C09107=1084.356,267.374,417.952,175.889,23.890,153.904
C09108=1084.350,267.126,417.980,175.886,23.886,153.903
C09109=1084.344,266.878,418.009,175.884,23.883,153.903
C09110=1084.339,266.630,418.037,175.881,23.880,153.903
C09111=1084.333,266.381,418.065,175.878,23.876,153.902
C09112=1084.328,266.133,418.094,175.876,23.873,153.902
C09113=1084.322,265.884,418.122,175.873,23.870,153.902
C09114=1084.317,265.636,418.151,175.870,23.867,153.901
C09115=1084.311,265.388,418.179,175.868,23.863,153.901
C09116=1084.305,265.140,418.207,175.865,23.860,153.901
C09117=1084.299,264.891,418.235,175.862,23.857,153.900
C09118=1084.294,264.643,418.263,175.860,23.854,153.900
C09119=1084.288,264.394,418.291,175.857,23.850,153.900
C09120=1084.283,264.146,418.319,175.854,23.847,153.899
C09121=1084.276,263.898,418.347,175.852,23.844,153.899
C09122=1084.270,263.649,418.376,175.848,23.841,153.899
C09123=1084.261,263.270,418.419,175.844,23.836,153.898
C09124=1084.253,262.891,418.461,175.840,23.831,153.898
C09125=1084.244,262.512,418.504,175.836,23.826,153.897
C09126=1084.234,262.133,418.546,175.831,23.821,153.897
C09127=1084.229,261.884,418.575,175.829,23.818,153.896
C09128=1084.223,261.636,418.603,175.826,23.815,153.896
C09129=1084.217,261.387,418.631,175.823,23.812,153.896
C09130=1084.211,261.140,418.658,175.821,23.809,153.895
C09131=1084.205,260.891,418.687,175.818,23.805,153.895
C09132=1084.200,260.643,418.715,175.816,23.802,153.895
C09133=1084.195,260.394,418.742,175.812,23.799,153.894
C09134=1084.188,260.146,418.770,175.809,23.796,153.894
C09135=1084.183,259.898,418.798,175.807,23.793,153.894
C09136=1084.177,259.649,418.826,175.804,23.790,153.893
C09137=1084.171,259.401,418.853,175.801,23.786,153.893
C09138=1084.165,259.152,418.882,175.799,23.783,153.893
C09139=1084.160,258.904,418.909,175.796,23.780,153.892
C09140=1084.153,258.655,418.937,175.793,23.777,153.892
C09141=1084.148,258.407,418.965,175.791,23.774,153.892
C09142=1084.142,258.159,418.993,175.788,23.770,153.891
C09143=1084.136,257.910,419.020,175.786,23.768,153.891
C09144=1084.131,257.662,419.048,175.782,23.764,153.891
C09145=1084.125,257.413,419.076,175.780,23.761,153.890
C09146=1084.119,257.165,419.102,175.777,23.758,153.890
C09147=1084.114,256.917,419.130,175.774,23.755,153.890
C09148=1084.108,256.668,419.159,175.771,23.751,153.889
C09149=1084.102,256.420,419.185,175.769,23.749,153.889
C09150=1084.097,256.172,419.213,175.766,23.745,153.889
C09151=1084.091,255.923,419.242,175.764,23.742,153.888
C09152=1084.085,255.675,419.268,175.761,23.739,153.888
C09153=1084.080,255.427,419.296,175.758,23.736,153.888
C09154=1084.074,255.177,419.324,175.756,23.732,153.887
C09155=1084.068,254.929,419.351,175.753,23.729,153.887
C09156=1084.063,254.681,419.379,175.750,23.726,153.887
C09157=1084.056,254.432,419.406,175.748,23.723,153.886
C09158=1084.051,254.184,419.434,175.744,23.720,153.886
C09159=1084.046,253.936,419.461,175.742,23.717,153.886
C09160=1084.039,253.687,419.489,175.739,23.713,153.885
C09161=1084.034,253.439,419.516,175.736,23.710,153.885
C09162=1084.028,253.190,419.543,175.734,23.707,153.885
C09163=1084.023,252.942,419.571,175.731,23.703,153.884
C09164=1084.017,252.693,419.598,175.729,23.701,153.884
C09165=1084.011,252.445,419.626,175.726,23.698,153.884
C09166=1084.006,252.196,419.653,175.723,23.694,153.883
C09167=1084.000,251.949,419.681,175.721,23.691,153.883
C09168=1083.994,251.699,419.708,175.718,23.688,153.883
C09169=1083.989,251.451,419.735,175.716,23.685,153.882
C09170=1083.983,251.203,419.763,175.713,23.681,153.882
C09171=1083.978,250.954,419.789,175.710,23.679,153.882
C09172=1083.973,250.706,419.817,175.708,23.675,153.881
C09173=1083.966,250.457,419.844,175.704,23.672,153.881
C09174=1083.961,250.209,419.872,175.702,23.669,153.881
C09175=1083.952,249.827,419.913,175.698,23.664,153.880
C09176=1083.944,249.445,419.955,175.694,23.659,153.880
C09177=1083.935,249.063,419.997,175.690,23.654,153.879
C09178=1083.926,248.682,420.039,175.686,23.649,153.879
C09179=1083.921,248.433,420.066,175.683,23.646,153.878
C09180=1083.915,248.185,420.093,175.681,23.643,153.878
C09181=1083.910,247.936,420.120,175.678,23.640,153.878
C09182=1083.905,247.687,420.147,175.676,23.636,153.877
C09183=1083.899,247.438,420.174,175.673,23.633,153.877
C09184=1083.893,247.190,420.202,175.670,23.630,153.877
C09185=1083.888,246.942,420.229,175.668,23.627,153.876
C09186=1083.882,246.693,420.255,175.665,23.623,153.876
C09187=1083.876,246.445,420.282,175.662,23.621,153.876
C09188=1083.871,246.196,420.309,175.659,23.617,153.875
C09189=1083.865,245.948,420.336,175.657,23.614,153.875
C09190=1083.859,245.699,420.363,175.654,23.611,153.875
C09191=1083.853,245.451,420.390,175.652,23.608,153.874
C09192=1083.848,245.202,420.417,175.649,23.605,153.874
C09193=1083.842,244.953,420.444,175.646,23.602,153.874
C09194=1083.837,244.705,420.470,175.644,23.598,153.873
C09195=1083.831,244.457,420.497,175.641,23.595,153.873
C09196=1083.826,244.208,420.524,175.639,23.592,153.873
C09197=1083.820,243.960,420.551,175.636,23.589,153.872
C09198=1083.814,243.711,420.577,175.634,23.586,153.872
C09199=1083.809,243.463,420.605,175.630,23.583,153.872
C09200=1083.804,243.214,420.631,175.628,23.580,153.871
C09201=1083.797,242.965,420.658,175.625,23.577,153.871
C09202=1083.791,242.717,420.685,175.623,23.573,153.871
C09203=1083.786,242.469,420.712,175.620,23.570,153.870
C09204=1083.780,242.220,420.738,175.618,23.567,153.870
C09205=1083.774,241.971,420.764,175.615,23.564,153.870
C09206=1083.769,241.723,420.791,175.613,23.561,153.869
C09207=1083.764,241.474,420.818,175.610,23.558,153.869
C09208=1083.758,241.226,420.845,175.607,23.555,153.869
C09209=1083.752,240.977,420.871,175.605,23.552,153.869
C09210=1083.746,240.729,420.898,175.602,23.548,153.868
C09211=1083.741,240.480,420.924,175.599,23.546,153.868
C09212=1083.735,240.232,420.951,175.596,23.542,153.868
C09213=1083.729,239.983,420.977,175.594,23.539,153.867
C09214=1083.723,239.735,421.004,175.591,23.536,153.867
C09215=1083.718,239.486,421.030,175.589,23.533,153.867
C09216=1083.712,239.238,421.057,175.586,23.530,153.866
C09217=1083.706,238.989,421.083,175.584,23.527,153.866
C09218=1083.701,238.740,421.109,175.581,23.524,153.866
C09219=1083.695,238.492,421.136,175.579,23.521,153.865
C09220=1083.689,238.244,421.162,175.576,23.517,153.865
C09221=1083.684,237.995,421.188,175.573,23.515,153.865
C09222=1083.678,237.746,421.215,175.571,23.511,153.864
C09223=1083.672,237.498,421.242,175.568,23.508,153.864
C09224=1083.667,237.249,421.268,175.565,23.505,153.864
C09225=1083.661,237.001,421.294,175.563,23.502,153.864
C09226=1083.656,236.752,421.320,175.560,23.499,153.863
C09227=1083.646,236.364,421.361,175.556,23.494,153.863
C09228=1083.638,235.975,421.403,175.552,23.489,153.862
C09229=1083.629,235.586,421.444,175.548,23.485,153.862
C09230=1083.620,235.197,421.484,175.545,23.480,153.861
C09231=1083.614,234.949,421.511,175.542,23.477,153.861
C09232=1083.609,234.700,421.537,175.540,23.474,153.861
C09233=1083.603,234.451,421.563,175.537,23.470,153.860
C09234=1083.597,234.202,421.589,175.534,23.467,153.860
C09235=1083.592,233.953,421.615,175.531,23.464,153.860
C09236=1083.586,233.705,421.642,175.529,23.461,153.859
C09237=1083.580,233.456,421.667,175.526,23.458,153.859
C09238=1083.574,233.208,421.694,175.524,23.455,153.859
C09239=1083.569,232.960,421.720,175.521,23.452,153.858
C09240=1083.564,232.711,421.745,175.519,23.449,153.858
C09241=1083.558,232.462,421.772,175.516,23.446,153.858
C09242=1083.552,232.214,421.797,175.514,23.443,153.858
C09243=1083.546,231.965,421.824,175.511,23.439,153.857
C09244=1083.541,231.716,421.850,175.509,23.436,153.857
C09245=1083.535,231.467,421.876,175.506,23.434,153.857
C09246=1083.530,231.219,421.902,175.504,23.430,153.856
C09247=1083.524,230.971,421.928,175.501,23.427,153.856
C09248=1083.518,230.722,421.954,175.498,23.424,153.856
C09249=1083.513,230.473,421.979,175.496,23.421,153.855
C09250=1083.507,230.225,422.006,175.493,23.418,153.855
C09251=1083.501,229.976,422.031,175.491,23.415,153.855
C09252=1083.496,229.728,422.057,175.488,23.412,153.854
C09253=1083.490,229.479,422.082,175.486,23.409,153.854
C09254=1083.484,229.230,422.108,175.484,23.406,153.854
C09255=1083.479,228.982,422.135,175.481,23.403,153.853
C09256=1083.472,228.733,422.160,175.478,23.400,153.853
C09257=1083.467,228.484,422.186,175.475,23.397,153.853
C09258=1083.461,228.236,422.211,175.473,23.393,153.852
C09259=1083.456,227.987,422.237,175.470,23.390,153.852
C09260=1083.450,227.739,422.262,175.468,23.388,153.852
C09261=1083.444,227.490,422.288,175.465,23.384,153.852
C09262=1083.439,227.241,422.314,175.463,23.381,153.851
C09263=1083.433,226.993,422.340,175.461,23.378,153.851
C09264=1083.427,226.744,422.366,175.458,23.375,153.851
C09265=1083.421,226.496,422.391,175.456,23.372,153.850
C09266=1083.416,226.247,422.417,175.453,23.369,153.850
C09267=1083.410,225.999,422.442,175.450,23.366,153.850
C09268=1083.405,225.750,422.468,175.447,23.363,153.850
C09269=1083.398,225.501,422.493,175.445,23.360,153.849
C09270=1083.393,225.252,422.519,175.443,23.357,153.849
C09271=1083.388,225.004,422.545,175.440,23.354,153.849
C09272=1083.382,224.755,422.570,175.438,23.351,153.848
C09273=1083.376,224.506,422.596,175.435,23.347,153.848
C09274=1083.371,224.258,422.621,175.433,23.345,153.848
C09275=1083.365,224.009,422.647,175.431,23.342,153.847
C09276=1083.359,223.761,422.672,175.428,23.338,153.847
C09277=1083.354,223.512,422.697,175.426,23.335,153.847
C09278=1083.348,223.263,422.723,175.423,23.332,153.846
C09279=1083.339,222.866,422.764,175.419,23.327,153.846
C09280=1083.330,222.468,422.804,175.416,23.323,153.845
C09281=1083.321,222.071,422.845,175.411,23.318,153.845
C09282=1083.313,221.674,422.885,175.407,23.313,153.844
C09283=1083.306,221.425,422.910,175.404,23.309,153.844
C09284=1083.301,221.177,422.935,175.402,23.306,153.844
C09285=1083.295,220.928,422.961,175.399,23.303,153.843
C09286=1083.289,220.679,422.986,175.397,23.301,153.843
C09287=1083.283,220.430,423.011,175.395,23.298,153.843
C09288=1083.278,220.182,423.037,175.392,23.294,153.842
C09289=1083.272,219.933,423.062,175.390,23.291,153.842
C09290=1083.267,219.685,423.086,175.388,23.289,153.842
C09291=1083.261,219.436,423.112,175.385,23.285,153.842
C09292=1083.255,219.187,423.138,175.383,23.282,153.841
C09293=1083.250,218.938,423.162,175.379,23.279,153.841
C09294=1083.244,218.690,423.187,175.377,23.276,153.841
C09295=1083.237,218.441,423.213,175.375,23.273,153.840
C09296=1083.233,218.192,423.237,175.372,23.270,153.840
C09297=1083.227,217.944,423.263,175.370,23.267,153.840
C09298=1083.221,217.696,423.288,175.368,23.264,153.839
C09299=1083.215,217.446,423.312,175.365,23.261,153.839
C09300=1083.210,217.198,423.338,175.363,23.258,153.839
C09301=1083.204,216.949,423.363,175.360,23.255,153.839
C09302=1083.198,216.700,423.388,175.358,23.252,153.838
C09303=1083.193,216.451,423.412,175.355,23.249,153.838
C09304=1083.187,216.203,423.438,175.353,23.245,153.838
C09305=1083.182,215.955,423.463,175.350,23.243,153.837
C09306=1083.176,215.705,423.488,175.348,23.240,153.837
C09307=1083.170,215.457,423.513,175.345,23.237,153.837
C09308=1083.164,215.208,423.537,175.343,23.234,153.836
C09309=1083.159,214.960,423.562,175.341,23.231,153.836
C09310=1083.154,214.710,423.587,175.338,23.228,153.836
C09311=1083.148,214.462,423.612,175.336,23.224,153.835
C09312=1083.142,214.213,423.637,175.334,23.222,153.835
C09313=1083.137,213.965,423.661,175.331,23.218,153.835
C09314=1083.131,213.716,423.687,175.329,23.215,153.834
C09315=1083.126,213.467,423.712,175.327,23.212,153.834
C09316=1083.120,213.218,423.737,175.324,23.209,153.834
C09317=1083.115,212.970,423.761,175.321,23.206,153.834
C09318=1083.109,212.720,423.786,175.318,23.203,153.833
C09319=1083.103,212.473,423.811,175.316,23.200,153.833
C09320=1083.097,212.223,423.835,175.314,23.197,153.833
C09321=1083.092,211.975,423.860,175.311,23.194,153.832
C09322=1083.086,211.726,423.885,175.309,23.191,153.832
C09323=1083.080,211.477,423.909,175.307,23.188,153.832
C09324=1083.075,211.228,423.934,175.304,23.185,153.831
C09325=1083.069,210.980,423.959,175.302,23.181,153.831
C09326=1083.064,210.732,423.983,175.300,23.179,153.831
C09327=1083.058,210.482,424.008,175.297,23.176,153.830
C09328=1083.052,210.234,424.032,175.294,23.173,153.830
C09329=1083.046,209.985,424.057,175.292,23.170,153.830
C09330=1083.041,209.736,424.082,175.290,23.167,153.829
C09331=1083.031,209.343,424.120,175.286,23.162,153.829
C09332=1083.023,208.950,424.159,175.282,23.157,153.829
C09333=1083.014,208.556,424.198,175.279,23.152,153.828
C09334=1083.005,208.163,424.236,175.275,23.148,153.828
C09335=1082.982,207.132,424.336,175.184,23.100,153.830
C09336=1082.976,206.884,424.359,175.181,23.097,153.830
C09337=1082.970,206.635,424.384,175.179,23.095,153.830
C09338=1082.965,206.386,424.408,175.177,23.093,153.830
C09339=1082.959,206.137,424.431,175.174,23.091,153.830
C09340=1082.954,205.889,424.456,175.172,23.089,153.830
C09341=1082.948,205.640,424.480,175.169,23.087,153.830
C09342=1082.943,205.391,424.503,175.167,23.085,153.830
C09343=1082.937,205.142,424.527,175.164,23.083,153.829
C09344=1082.931,204.894,424.551,175.161,23.080,153.829
C09345=1082.926,204.644,424.575,175.159,23.079,153.829
C09346=1082.921,204.396,424.599,175.156,23.076,153.829
C09347=1082.914,204.148,424.623,175.154,23.075,153.829
C09348=1082.909,203.898,424.646,175.152,23.072,153.829
C09349=1082.904,203.649,424.671,175.149,23.070,153.829
C09350=1082.898,203.400,424.694,175.147,23.068,153.829
C09351=1082.893,203.152,424.718,175.144,23.066,153.829
C09352=1082.887,202.903,424.742,175.142,23.064,153.829
C09353=1082.882,202.654,424.765,175.139,23.062,153.829
C09354=1082.875,202.406,424.789,175.136,23.060,153.828
C09355=1082.871,202.157,424.812,175.134,23.058,153.828
C09356=1082.864,201.908,424.836,175.131,23.056,153.828
C09357=1082.859,201.658,424.860,175.129,23.054,153.828
C09358=1082.853,201.410,424.884,175.127,23.052,153.828
C09359=1082.847,201.161,424.906,175.124,23.050,153.828
C09360=1082.842,200.913,424.931,175.122,23.048,153.828
C09361=1082.836,200.664,424.954,175.119,23.046,153.828
C09362=1082.830,200.414,424.978,175.117,23.044,153.828
C09363=1082.824,200.166,425.001,175.115,23.042,153.828
C09364=1082.818,199.917,425.025,175.112,23.040,153.828
C09365=1082.813,199.668,425.048,175.109,23.037,153.828
C09366=1082.808,199.419,425.071,175.106,23.035,153.828
C09367=1082.802,199.171,425.095,175.104,23.033,153.827
C09368=1082.797,198.922,425.119,175.101,23.031,153.827
C09369=1082.791,198.673,425.142,175.099,23.029,153.827
C09370=1082.785,198.425,425.165,175.097,23.027,153.827
C09371=1082.779,198.175,425.189,175.094,23.025,153.827
C09372=1082.773,197.926,425.213,175.092,23.023,153.827
C09373=1082.768,197.677,425.236,175.089,23.021,153.827
C09374=1082.763,197.428,425.259,175.087,23.019,153.827
C09375=1082.756,197.180,425.283,175.085,23.017,153.827
C09376=1082.751,196.931,425.306,175.082,23.015,153.827
C09377=1082.746,196.682,425.329,175.080,23.013,153.827
C09378=1082.740,196.434,425.353,175.077,23.011,153.827
C09379=1082.734,196.185,425.376,175.075,23.009,153.826
C09380=1082.729,195.935,425.400,175.072,23.007,153.826
C09381=1082.723,195.687,425.422,175.070,23.005,153.826
C09382=1082.717,195.438,425.446,175.068,23.003,153.826
C09383=1082.712,195.189,425.469,175.065,23.001,153.826
C09384=1082.707,194.940,425.493,175.063,22.999,153.826
C09385=1082.701,194.691,425.516,175.060,22.997,153.826
C09386=1082.695,194.443,425.539,175.057,22.994,153.826
C09387=1082.690,194.194,425.563,175.055,22.992,153.826
C09388=1082.684,193.945,425.586,175.052,22.990,153.826
C09389=1082.678,193.696,425.609,175.050,22.988,153.826
C09390=1082.673,193.447,425.632,175.048,22.986,153.825
C09391=1082.668,193.198,425.655,175.045,22.984,153.825
C09392=1082.662,192.950,425.679,175.043,22.982,153.825
C09393=1082.656,192.701,425.702,175.040,22.980,153.825
C09394=1082.650,192.452,425.725,175.038,22.978,153.825
C09395=1082.645,192.203,425.748,175.036,22.976,153.825
C09396=1082.638,191.924,425.773,175.033,22.974,153.825
C09397=1082.632,191.645,425.800,175.031,22.972,153.825
C09398=1082.626,191.366,425.825,175.028,22.969,153.825
C09399=1082.620,191.087,425.851,175.025,22.967,153.825
C09400=1082.614,190.838,425.874,175.023,22.965,153.825
C09401=1082.609,190.589,425.898,175.020,22.963,153.824
C09402=1082.604,190.340,425.920,175.018,22.961,153.824
C09403=1082.598,190.091,425.943,175.016,22.959,153.824
C09404=1082.592,189.842,425.966,175.013,22.956,153.824
C09405=1082.587,189.594,425.989,175.011,22.955,153.824
C09406=1082.582,189.344,426.012,175.008,22.952,153.824
C09407=1082.576,189.096,426.035,175.006,22.950,153.824
C09408=1082.571,188.847,426.058,175.004,22.948,153.824
C09409=1082.565,188.598,426.081,175.001,22.946,153.824
C09410=1082.559,188.349,426.104,174.999,22.944,153.823
C09411=1082.554,188.100,426.128,174.996,22.942,153.823
C09412=1082.549,187.851,426.150,174.994,22.940,153.823
C09413=1082.543,187.603,426.173,174.992,22.938,153.823
C09414=1082.537,187.354,426.196,174.989,22.936,153.823
C09415=1082.532,187.105,426.219,174.987,22.934,153.823
C09416=1082.526,186.856,426.242,174.984,22.932,153.823
C09417=1082.521,186.607,426.264,174.982,22.929,153.823
C09418=1082.516,186.358,426.288,174.980,22.927,153.823
C09419=1082.510,186.109,426.311,174.977,22.925,153.823
C09420=1082.505,185.860,426.333,174.975,22.923,153.823
C09421=1082.499,185.611,426.356,174.973,22.921,153.822
C09422=1082.494,185.363,426.379,174.970,22.919,153.822
C09423=1082.488,185.113,426.401,174.968,22.917,153.822
C09424=1082.483,184.865,426.424,174.966,22.915,153.822
C09425=1082.477,184.616,426.447,174.964,22.913,153.822
C09426=1082.471,184.367,426.470,174.962,22.911,153.822
C09427=1082.466,184.117,426.492,174.959,22.909,153.822
C09428=1082.459,183.869,426.515,174.957,22.907,153.822
C09429=1082.454,183.620,426.537,174.954,22.905,153.822
C09430=1082.449,183.372,426.560,174.952,22.903,153.822
C09431=1082.443,183.122,426.582,174.949,22.901,153.822
C09432=1082.437,182.873,426.605,174.947,22.899,153.822
C09433=1082.431,182.625,426.628,174.945,22.897,153.821
C09434=1082.425,182.375,426.650,174.942,22.895,153.821
C09435=1082.420,182.126,426.673,174.940,22.893,153.821
C09436=1082.414,181.878,426.695,174.937,22.891,153.821
C09437=1082.408,181.629,426.717,174.935,22.889,153.821
C09438=1082.403,181.380,426.740,174.933,22.887,153.821
C09439=1082.397,181.131,426.763,174.931,22.885,153.821
C09440=1082.391,180.882,426.785,174.929,22.884,153.821
C09441=1082.385,180.633,426.808,174.926,22.881,153.821
C09442=1082.380,180.384,426.829,174.924,22.880,153.821
C09443=1082.374,180.135,426.852,174.921,22.877,153.821
C09444=1082.368,179.886,426.874,174.919,22.875,153.821
C09445=1082.363,179.637,426.897,174.917,22.873,153.820
C09446=1082.357,179.388,426.920,174.914,22.871,153.820
C09447=1082.351,179.140,426.941,174.912,22.869,153.820
C09448=1082.346,178.891,426.964,174.909,22.867,153.820
C09449=1082.340,178.641,426.986,174.907,22.865,153.820
C09450=1082.334,178.393,427.009,174.905,22.864,153.820
C09451=1082.329,178.144,427.031,174.903,22.861,153.820
C09452=1082.323,177.895,427.054,174.901,22.860,153.820
C09453=1082.317,177.646,427.075,174.898,22.857,153.820
C09454=1082.311,177.397,427.098,174.896,22.856,153.820
C09455=1082.306,177.148,427.120,174.893,22.853,153.820
C09456=1082.300,176.899,427.142,174.891,22.851,153.819
C09457=1082.295,176.650,427.165,174.889,22.849,153.819
C09458=1082.290,176.401,427.186,174.886,22.847,153.819
C09459=1082.283,176.153,427.209,174.884,22.845,153.819
C09460=1082.277,175.872,427.234,174.882,22.843,153.819
C09461=1082.271,175.593,427.259,174.879,22.841,153.819
C09462=1082.265,175.314,427.283,174.877,22.838,153.819
C09463=1082.258,175.035,427.309,174.874,22.837,153.819
C09464=1082.252,174.786,427.330,174.872,22.834,153.819
C09465=1082.247,174.537,427.352,174.870,22.832,153.819
C09466=1082.242,174.288,427.375,174.867,22.830,153.819
C09467=1082.236,174.039,427.397,174.865,22.828,153.818
C09468=1082.231,173.790,427.419,174.862,22.826,153.818
C09469=1082.225,173.541,427.440,174.860,22.824,153.818
C09470=1082.219,173.292,427.463,174.858,22.822,153.818
C09471=1082.214,173.043,427.485,174.856,22.820,153.818
C09472=1082.208,172.794,427.507,174.854,22.818,153.818
C09473=1082.202,172.545,427.530,174.851,22.816,153.818
C09474=1082.197,172.297,427.551,174.849,22.814,153.818
C09475=1082.191,172.047,427.573,174.847,22.812,153.818
C09476=1082.186,171.798,427.595,174.844,22.810,153.818
C09477=1082.180,171.549,427.617,174.842,22.808,153.817
C09478=1082.174,171.300,427.640,174.841,22.806,153.817
C09479=1082.169,171.052,427.661,174.838,22.804,153.817
C09480=1082.163,170.802,427.683,174.836,22.802,153.817
C09481=1082.158,170.554,427.705,174.833,22.799,153.817
C09482=1082.152,170.304,427.727,174.831,22.798,153.817
C09483=1082.147,170.056,427.749,174.829,22.795,153.817
C09484=1082.141,169.807,427.771,174.827,22.794,153.817
C09485=1082.136,169.557,427.793,174.825,22.792,153.817
C09486=1082.130,169.309,427.814,174.822,22.790,153.817
C09487=1082.125,169.059,427.837,174.820,22.787,153.816
C09488=1082.119,168.811,427.858,174.818,22.785,153.816
C09489=1082.114,168.561,427.880,174.815,22.783,153.816
C09490=1082.108,168.313,427.901,174.814,22.781,153.816
C09491=1082.103,168.063,427.924,174.811,22.779,153.816
C09492=1082.097,167.815,427.946,174.809,22.777,153.816
C09493=1082.091,167.566,427.968,174.807,22.775,153.816
C09494=1082.086,167.317,427.989,174.804,22.773,153.816
C09495=1082.080,167.068,428.011,174.802,22.771,153.816
C09496=1082.075,166.819,428.033,174.800,22.769,153.815
C09497=1082.069,166.570,428.055,174.798,22.767,153.815
C09498=1082.064,166.321,428.076,174.796,22.764,153.815
C09499=1082.058,166.072,428.098,174.793,22.763,153.815
C09500=1082.053,165.823,428.120,174.791,22.760,153.815
C09501=1082.048,165.574,428.142,174.790,22.759,153.815
C09502=1082.042,165.325,428.163,174.787,22.756,153.815
C09503=1082.037,165.076,428.185,174.785,22.754,153.815
C09504=1082.031,164.826,428.206,174.782,22.752,153.815
C09505=1082.026,164.578,428.228,174.780,22.750,153.814
C09506=1082.020,164.328,428.249,174.779,22.748,153.814
C09507=1082.015,164.080,428.271,174.776,22.746,153.814
C09508=1082.009,163.830,428.293,174.774,22.744,153.814
C09509=1082.004,163.582,428.315,174.772,22.742,153.814
C09510=1081.999,163.333,428.336,174.769,22.739,153.814
C09511=1081.993,163.084,428.358,174.768,22.737,153.814
C09512=1081.988,162.835,428.380,174.766,22.735,153.813
C09513=1081.982,162.585,428.400,174.763,22.733,153.813
C09514=1081.977,162.336,428.422,174.761,22.731,153.813
C09515=1081.972,162.088,428.444,174.758,22.729,153.813
C09516=1081.966,161.838,428.466,174.757,22.727,153.813
C09517=1081.961,161.590,428.487,174.755,22.725,153.813
C09518=1081.955,161.341,428.509,174.752,22.723,153.813
C09519=1081.950,161.091,428.530,174.750,22.721,153.813
C09520=1081.944,160.842,428.552,174.748,22.718,153.813
C09521=1081.938,160.594,428.573,174.746,22.717,153.812
C09522=1081.933,160.345,428.594,174.744,22.715,153.812
C09523=1081.927,160.095,428.615,174.741,22.712,153.812
C09524=1081.920,159.815,428.639,174.739,22.710,153.812
C09525=1081.915,159.536,428.663,174.737,22.708,153.812
C09526=1081.908,159.256,428.687,174.735,22.705,153.812
C09527=1081.902,158.977,428.711,174.732,22.704,153.812
C09528=1081.896,158.727,428.732,174.730,22.701,153.812
C09529=1081.891,158.479,428.754,174.727,22.699,153.811
C09530=1081.884,158.230,428.775,174.725,22.697,153.811
C09531=1081.879,157.980,428.796,174.723,22.695,153.811
C09532=1081.874,157.732,428.818,174.721,22.693,153.811
C09533=1081.868,157.482,428.839,174.719,22.691,153.811
C09534=1081.863,157.233,428.860,174.716,22.689,153.811
C09535=1081.857,156.984,428.881,174.715,22.687,153.811
C09536=1081.852,156.735,428.902,174.713,22.685,153.811
C09537=1081.846,156.486,428.923,174.710,22.683,153.811
C09538=1081.840,156.237,428.945,174.708,22.681,153.811
C09539=1081.835,155.988,428.965,174.706,22.679,153.810
C09540=1081.829,155.740,428.987,174.704,22.677,153.810
C09541=1081.823,155.490,429.008,174.702,22.674,153.810
C09542=1081.818,155.241,429.029,174.699,22.673,153.810
C09543=1081.812,154.992,429.049,174.698,22.671,153.810
C09544=1081.806,154.743,429.071,174.696,22.668,153.810
C09545=1081.801,154.494,429.092,174.693,22.666,153.810
C09546=1081.795,154.245,429.113,174.691,22.664,153.810
C09547=1081.789,153.996,429.135,174.689,22.663,153.809
C09548=1081.784,153.747,429.155,174.687,22.660,153.809
C09549=1081.778,153.497,429.176,174.685,22.658,153.809
C09550=1081.773,153.249,429.197,174.682,22.656,153.809
C09551=1081.767,153.000,429.218,174.681,22.654,153.809
C09552=1081.761,152.750,429.239,174.679,22.652,153.809
C09553=1081.756,152.501,429.260,174.676,22.650,153.809
C09554=1081.750,152.253,429.281,174.675,22.648,153.809
C09555=1081.745,152.004,429.302,174.672,22.646,153.808
C09556=1081.739,151.754,429.324,174.670,22.644,153.808
C09557=1081.734,151.505,429.344,174.668,22.641,153.808
C09558=1081.728,151.256,429.365,174.666,22.640,153.808
C09559=1081.722,151.007,429.386,174.664,22.638,153.808
C09560=1081.717,150.758,429.407,174.662,22.635,153.808
C09561=1081.711,150.509,429.428,174.660,22.634,153.808
C09562=1081.706,150.260,429.449,174.658,22.631,153.808
C09563=1081.700,150.010,429.470,174.656,22.629,153.807
C09564=1081.695,149.762,429.491,174.653,22.627,153.807
C09565=1081.689,149.513,429.511,174.652,22.625,153.807
C09566=1081.683,149.264,429.531,174.649,22.623,153.807
C09567=1081.677,149.015,429.553,174.647,22.621,153.807
C09568=1081.672,148.766,429.574,174.646,22.619,153.807
C09569=1081.667,148.516,429.594,174.643,22.617,153.807
C09570=1081.662,148.267,429.615,174.641,22.615,153.807
C09571=1081.655,148.018,429.636,174.639,22.612,153.807
C09572=1081.649,147.769,429.656,174.637,22.611,153.806
C09573=1081.644,147.520,429.677,174.635,22.608,153.806
C09574=1081.639,147.271,429.697,174.632,22.607,153.806
C09575=1081.633,147.022,429.719,174.631,22.605,153.806
C09576=1081.627,146.773,429.739,174.629,22.602,153.806
C09577=1081.621,146.524,429.759,174.626,22.600,153.806
C09578=1081.616,146.275,429.780,174.625,22.599,153.806
C09579=1081.610,146.025,429.801,174.622,22.596,153.806
C09580=1081.604,145.777,429.822,174.620,22.594,153.805
C09581=1081.599,145.528,429.842,174.619,22.592,153.805
C09582=1081.594,145.279,429.863,174.616,22.590,153.805
C09583=1081.588,145.029,429.883,174.614,22.588,153.805
C09584=1081.582,144.780,429.904,174.613,22.586,153.805
C09585=1081.576,144.531,429.924,174.610,22.584,153.805
C09586=1081.571,144.282,429.945,174.608,22.582,153.805
C09587=1081.565,144.033,429.965,174.606,22.580,153.804
C09588=1081.559,143.753,429.988,174.604,22.577,153.804
C09589=1081.552,143.473,430.011,174.602,22.575,153.804
C09590=1081.546,143.193,430.035,174.600,22.573,153.804
C09591=1081.540,142.914,430.058,174.597,22.571,153.804
C09592=1081.535,142.664,430.078,174.595,22.568,153.804
C09593=1081.529,142.415,430.099,174.593,22.566,153.804
C09594=1081.523,142.166,430.119,174.591,22.564,153.803
C09595=1081.517,141.917,430.140,174.589,22.562,153.803
C09596=1081.512,141.668,430.160,174.587,22.559,153.803
C09597=1081.506,141.419,430.180,174.585,22.558,153.803
C09598=1081.501,141.170,430.201,174.583,22.556,153.803
C09599=1081.496,140.920,430.221,174.580,22.553,153.803
C09600=1081.490,140.672,430.241,174.579,22.552,153.803
C09601=1081.484,140.423,430.262,174.577,22.549,153.803
C09602=1081.478,140.173,430.282,174.574,22.547,153.802
C09603=1081.473,139.924,430.303,174.573,22.545,153.802
C09604=1081.467,139.675,430.323,174.571,22.543,153.802
C09605=1081.461,139.426,430.343,174.568,22.541,153.802
C09606=1081.456,139.176,430.363,174.567,22.539,153.802
C09607=1081.450,138.927,430.383,174.565,22.537,153.802
C09608=1081.445,138.678,430.404,174.562,22.535,153.802
C09609=1081.439,138.429,430.424,174.561,22.533,153.801
C09610=1081.433,138.180,430.444,174.559,22.530,153.801
C09611=1081.427,137.931,430.464,174.556,22.528,153.801
C09612=1081.422,137.682,430.485,174.555,22.526,153.801
C09613=1081.416,137.433,430.505,174.552,22.524,153.801
C09614=1081.411,137.183,430.525,174.551,22.522,153.801
C09615=1081.405,136.934,430.545,174.549,22.520,153.801
C09616=1081.400,136.685,430.565,174.546,22.518,153.801
C09617=1081.394,136.436,430.585,174.545,22.516,153.800
C09618=1081.389,136.187,430.606,174.543,22.514,153.800
C09619=1081.383,135.938,430.626,174.540,22.511,153.800
C09620=1081.378,135.689,430.646,174.539,22.509,153.800
C09621=1081.372,135.440,430.666,174.537,22.507,153.800
C09622=1081.365,135.190,430.686,174.534,22.505,153.800
C09623=1081.360,134.941,430.706,174.533,22.503,153.799
C09624=1081.354,134.692,430.726,174.530,22.501,153.799
C09625=1081.349,134.443,430.746,174.529,22.499,153.799
C09626=1081.343,134.194,430.766,174.527,22.497,153.799
C09627=1081.338,133.945,430.787,174.524,22.495,153.799
C09628=1081.332,133.695,430.806,174.523,22.493,153.799
C09629=1081.326,133.447,430.826,174.521,22.490,153.799
C09630=1081.321,133.197,430.846,174.519,22.489,153.799
C09631=1081.315,132.948,430.866,174.517,22.486,153.798
C09632=1081.310,132.699,430.886,174.515,22.484,153.798
C09633=1081.304,132.450,430.906,174.513,22.482,153.798
C09634=1081.298,132.201,430.925,174.511,22.480,153.798
C09635=1081.293,131.951,430.946,174.509,22.477,153.798
C09636=1081.287,131.703,430.966,174.507,22.476,153.798
C09637=1081.281,131.453,430.985,174.505,22.473,153.797
C09638=1081.275,131.204,431.005,174.504,22.471,153.797
C09639=1081.270,130.955,431.026,174.501,22.470,153.797
C09640=1081.264,130.706,431.045,174.499,22.467,153.797
C09641=1081.258,130.457,431.065,174.498,22.465,153.797
C09642=1081.252,130.208,431.084,174.495,22.463,153.797
C09643=1081.246,129.959,431.104,174.494,22.461,153.797
C09644=1081.241,129.710,431.125,174.492,22.459,153.797
C09645=1081.236,129.460,431.144,174.489,22.457,153.796
C09646=1081.230,129.211,431.164,174.488,22.455,153.796
C09647=1081.224,128.962,431.183,174.486,22.452,153.796
C09648=1081.218,128.713,431.203,174.484,22.450,153.796
C09649=1081.212,128.464,431.222,174.482,22.448,153.796
C09650=1081.207,128.215,431.243,174.480,22.446,153.796
C09651=1081.201,127.965,431.262,174.478,22.445,153.796
C09652=1081.195,127.685,431.284,174.476,22.442,153.795
C09653=1081.188,127.405,431.306,174.474,22.439,153.795
C09654=1081.182,127.125,431.328,174.471,22.437,153.795
C09655=1081.175,126.845,431.350,174.469,22.435,153.795
C09656=1081.169,126.596,431.370,174.468,22.433,153.795
C09657=1081.164,126.347,431.389,174.465,22.431,153.795
C09658=1081.159,126.098,431.410,174.464,22.429,153.794
C09659=1081.153,125.848,431.429,174.462,22.426,153.794
C09660=1081.147,125.599,431.449,174.459,22.424,153.794
C09661=1081.141,125.350,431.468,174.458,22.422,153.794
C09662=1081.135,125.101,431.488,174.456,22.420,153.794
C09663=1081.129,124.852,431.508,174.454,22.418,153.794
C09664=1081.124,124.602,431.527,174.452,22.416,153.794
C09665=1081.119,124.354,431.546,174.451,22.414,153.793
C09666=1081.113,124.105,431.566,174.448,22.411,153.793
C09667=1081.108,123.855,431.585,174.446,22.409,153.793
C09668=1081.102,123.606,431.605,174.445,22.407,153.793
C09669=1081.096,123.357,431.625,174.442,22.405,153.793
C09670=1081.090,123.107,431.644,174.441,22.403,153.793
C09671=1081.084,122.858,431.664,174.439,22.401,153.793
C09672=1081.079,122.609,431.683,174.437,22.399,153.792
C09673=1081.074,122.360,431.702,174.435,22.396,153.792
C09674=1081.068,122.111,431.721,174.434,22.394,153.792
C09675=1081.062,121.862,431.741,174.431,22.392,153.792
C09676=1081.056,121.613,431.760,174.429,22.389,153.792
C09677=1081.051,121.363,431.780,174.428,22.388,153.791
C09678=1081.045,121.114,431.799,174.425,22.385,153.791
C09679=1081.040,120.865,431.819,174.424,22.383,153.791
C09680=1081.035,120.616,431.838,174.422,22.381,153.791
C09681=1081.029,120.366,431.858,174.420,22.379,153.791
C09682=1081.023,120.117,431.877,174.418,22.377,153.791
C09683=1081.017,119.868,431.897,174.417,22.375,153.791
C09684=1081.011,119.619,431.916,174.415,22.372,153.790
C09685=1081.006,119.370,431.935,174.412,22.370,153.790
C09686=1081.001,119.121,431.954,174.411,22.368,153.790
C09687=1080.995,118.871,431.973,174.409,22.366,153.790
C09688=1080.989,118.622,431.993,174.407,22.364,153.790
C09689=1080.983,118.373,432.013,174.405,22.361,153.789
C09690=1080.978,118.124,432.032,174.403,22.359,153.789
C09691=1080.973,117.875,432.051,174.401,22.357,153.789
C09692=1080.967,117.625,432.070,174.400,22.355,153.789
C09693=1080.961,117.376,432.089,174.398,22.352,153.789
C09694=1080.956,117.127,432.108,174.396,22.350,153.789
C09695=1080.950,116.878,432.127,174.394,22.348,153.788
C09696=1080.945,116.628,432.147,174.393,22.346,153.788
C09697=1080.939,116.379,432.166,174.390,22.344,153.788
C09698=1080.934,116.130,432.185,174.388,22.341,153.788
C09699=1080.928,115.881,432.204,174.387,22.339,153.788
C09700=1080.922,115.632,432.224,174.385,22.337,153.788
C09701=1080.917,115.383,432.243,174.383,22.335,153.787
C09702=1080.911,115.134,432.262,174.381,22.333,153.787
C09703=1080.906,114.884,432.281,174.380,22.330,153.787
C09704=1080.900,114.635,432.301,174.377,22.328,153.787
C09705=1080.895,114.386,432.319,174.376,22.326,153.787
C09706=1080.889,114.137,432.339,174.374,22.324,153.786
C09707=1080.884,113.887,432.358,174.372,22.322,153.786
C09708=1080.878,113.639,432.376,174.370,22.319,153.786
C09709=1080.872,113.389,432.395,174.369,22.317,153.786
C09710=1080.866,113.140,432.415,174.366,22.315,153.786
C09711=1080.861,112.890,432.433,174.365,22.313,153.786
C09712=1080.856,112.641,432.452,174.363,22.311,153.785
C09713=1080.850,112.392,432.471,174.361,22.309,153.785
C09714=1080.844,112.143,432.490,174.359,22.306,153.785
C09715=1080.838,111.893,432.509,174.358,22.304,153.785
C09716=1080.831,111.614,432.531,174.356,22.302,153.785
C09717=1080.826,111.333,432.552,174.353,22.299,153.785
C09718=1080.819,111.053,432.573,174.351,22.296,153.784
C09719=1080.812,110.773,432.594,174.349,22.294,153.784
C09720=1080.807,110.524,432.613,174.348,22.292,153.784
C09721=1080.802,110.274,432.632,174.345,22.290,153.784
C09722=1080.795,110.025,432.650,174.344,22.288,153.784
C09723=1080.790,109.777,432.669,174.342,22.285,153.783
C09724=1080.784,109.527,432.688,174.340,22.283,153.783
C09725=1080.778,109.278,432.707,174.338,22.281,153.783
C09726=1080.772,109.029,432.726,174.337,22.279,153.783
C09727=1080.767,108.779,432.744,174.334,22.277,153.783
C09728=1080.761,108.530,432.763,174.333,22.275,153.783
C09729=1080.755,108.281,432.782,174.331,22.272,153.782
C09730=1080.750,108.032,432.801,174.330,22.270,153.782
C09731=1080.744,107.783,432.820,174.327,22.268,153.782
C09732=1080.739,107.533,432.838,174.326,22.266,153.782
C09733=1080.733,107.284,432.857,174.324,22.263,153.782
C09734=1080.727,107.035,432.876,174.322,22.262,153.782
C09735=1080.722,106.785,432.894,174.320,22.259,153.781
C09736=1080.716,106.536,432.913,174.319,22.257,153.781
C09737=1080.710,106.287,432.932,174.316,22.254,153.781
C09738=1080.704,106.039,432.950,174.315,22.253,153.781
C09739=1080.699,105.788,432.969,174.313,22.250,153.781
C09740=1080.693,105.539,432.988,174.312,22.248,153.780
C09741=1080.687,105.291,433.006,174.309,22.245,153.780
C09742=1080.682,105.041,433.025,174.308,22.244,153.780
C09743=1080.676,104.791,433.043,174.307,22.242,153.780
C09744=1080.671,104.543,433.062,174.304,22.239,153.780
C09745=1080.665,104.293,433.081,174.303,22.237,153.779
C09746=1080.659,104.044,433.099,174.301,22.235,153.779
C09747=1080.654,103.795,433.118,174.299,22.233,153.779
C09748=1080.648,103.546,433.136,174.297,22.230,153.779
C09749=1080.642,103.296,433.155,174.296,22.228,153.779
C09750=1080.636,103.047,433.173,174.294,22.226,153.779
C09751=1080.631,102.798,433.192,174.292,22.223,153.778
C09752=1080.626,102.548,433.211,174.290,22.221,153.778
C09753=1080.620,102.299,433.229,174.289,22.219,153.778
C09754=1080.614,102.050,433.248,174.286,22.217,153.778
C09755=1080.609,101.801,433.266,174.285,22.214,153.778
C09756=1080.603,101.552,433.285,174.283,22.212,153.777
C09757=1080.598,101.302,433.302,174.282,22.210,153.777
C09758=1080.592,101.053,433.322,174.279,22.207,153.777
C09759=1080.586,100.803,433.340,174.278,22.205,153.777
C09760=1080.580,100.555,433.358,174.276,22.203,153.777
C09761=1080.575,100.305,433.376,174.274,22.201,153.776
C09762=1080.569,100.056,433.395,174.273,22.199,153.776
C09763=1080.563,99.806,433.413,174.271,22.196,153.776
C09764=1080.557,99.557,433.432,174.270,22.194,153.776
C09765=1080.551,99.308,433.449,174.267,22.192,153.776
C09766=1080.546,99.059,433.469,174.266,22.190,153.776
C09767=1080.540,98.810,433.486,174.264,22.187,153.775
C09768=1080.534,98.561,433.505,174.262,22.185,153.775
C09769=1080.529,98.311,433.523,174.260,22.183,153.775
C09770=1080.523,98.061,433.541,174.259,22.181,153.775
C09771=1080.517,97.813,433.559,174.257,22.178,153.775
C09772=1080.512,97.563,433.578,174.255,22.176,153.774
C09773=1080.506,97.315,433.596,174.254,22.174,153.774
C09774=1080.500,97.065,433.614,174.252,22.172,153.774
C09775=1080.494,96.815,433.633,174.250,22.170,153.774
C09776=1080.489,96.566,433.651,174.248,22.167,153.774
C09777=1080.482,96.317,433.669,174.247,22.165,153.773
C09778=1080.478,96.067,433.687,174.245,22.163,153.773
C09779=1080.471,95.818,433.706,174.243,22.161,153.773
C09780=1080.465,95.539,433.726,174.241,22.158,153.773
C09781=1080.459,95.258,433.746,174.239,22.155,153.773
C09782=1080.453,94.978,433.766,174.238,22.153,153.772
C09783=1080.446,94.698,433.787,174.235,22.151,153.772
C09784=1080.441,94.449,433.805,174.233,22.148,153.772
C09785=1080.435,94.200,433.823,174.232,22.146,153.772
C09786=1080.429,93.951,433.841,174.231,22.144,153.772
C09787=1080.424,93.701,433.859,174.229,22.141,153.771
C09788=1080.418,93.452,433.877,174.227,22.139,153.771
C09789=1080.412,93.203,433.896,174.225,22.137,153.771
C09790=1080.406,92.953,433.913,174.224,22.134,153.771
C09791=1080.401,92.703,433.932,174.221,22.132,153.771
C09792=1080.395,92.454,433.949,174.220,22.130,153.770
C09793=1080.390,92.206,433.968,174.219,22.128,153.770
C09794=1080.384,91.956,433.986,174.217,22.125,153.770
C09795=1080.379,91.707,434.004,174.215,22.123,153.770
C09796=1080.373,91.457,434.022,174.213,22.121,153.770
C09797=1080.367,91.208,434.039,174.212,22.119,153.769
C09798=1080.362,90.959,434.058,174.210,22.116,153.769
C09799=1080.356,90.710,434.076,174.208,22.114,153.769
C09800=1080.350,90.461,434.094,174.207,22.112,153.769
C09801=1080.344,90.211,434.112,174.205,22.109,153.769
C09802=1080.339,89.962,434.129,174.203,22.107,153.768
C09803=1080.333,89.712,434.147,174.201,22.105,153.768
C09804=1080.327,89.463,434.165,174.200,22.103,153.768
C09805=1080.321,89.214,434.183,174.198,22.100,153.768
C09806=1080.315,88.965,434.201,174.196,22.098,153.768
C09807=1080.310,88.716,434.218,174.195,22.096,153.767
C09808=1080.303,88.466,434.236,174.193,22.094,153.767
C09809=1080.298,88.217,434.254,174.191,22.092,153.767
C09810=1080.292,87.967,434.272,174.189,22.089,153.767
C09811=1080.286,87.718,434.289,174.188,22.087,153.767
C09812=1080.280,87.469,434.307,174.187,22.085,153.766
C09813=1080.275,87.219,434.325,174.185,22.082,153.766
C09814=1080.270,86.970,434.343,174.183,22.080,153.766
C09815=1080.264,86.720,434.361,174.181,22.078,153.766
C09816=1080.258,86.471,434.379,174.180,22.075,153.766
C09817=1080.253,86.222,434.396,174.177,22.073,153.765
C09818=1080.247,85.973,434.414,174.176,22.071,153.765
C09819=1080.241,85.724,434.432,174.175,22.069,153.765
C09820=1080.235,85.474,434.450,174.173,22.066,153.765
C09821=1080.229,85.225,434.467,174.171,22.064,153.764
C09822=1080.224,84.976,434.485,174.169,22.062,153.764
C09823=1080.218,84.726,434.503,174.168,22.060,153.764
C09824=1080.212,84.477,434.520,174.167,22.057,153.764
C09825=1080.207,84.228,434.538,174.164,22.055,153.764
C09826=1080.201,83.978,434.556,174.163,22.052,153.763
C09827=1080.195,83.729,434.573,174.161,22.050,153.763
C09828=1080.190,83.480,434.591,174.159,22.048,153.763
C09829=1080.183,83.230,434.609,174.158,22.046,153.763
C09830=1080.178,82.981,434.626,174.156,22.043,153.763
C09831=1080.173,82.732,434.643,174.155,22.041,153.762
C09832=1080.167,82.483,434.661,174.153,22.039,153.762
C09833=1080.161,82.233,434.679,174.151,22.036,153.762
C09834=1080.156,81.984,434.696,174.150,22.034,153.762
C09835=1080.150,81.735,434.714,174.148,22.031,153.762
C09836=1080.143,81.485,434.731,174.146,22.029,153.761
C09837=1080.138,81.236,434.749,174.144,22.027,153.761
C09838=1080.132,80.987,434.766,174.143,22.025,153.761
C09839=1080.127,80.738,434.783,174.142,22.023,153.761
C09840=1080.121,80.488,434.801,174.140,22.020,153.760
C09841=1080.115,80.239,434.819,174.138,22.018,153.760
C09842=1080.110,79.990,434.836,174.136,22.015,153.760
C09843=1080.104,79.741,434.854,174.135,22.013,153.760
C09844=1080.098,79.460,434.874,174.133,22.010,153.760
C09845=1080.092,79.180,434.893,174.131,22.008,153.759
C09846=1080.085,78.900,434.912,174.129,22.005,153.759
C09847=1080.078,78.620,434.932,174.127,22.003,153.759
C09848=1080.073,78.371,434.949,174.126,22.000,153.759
C09849=1080.067,78.121,434.967,174.125,21.998,153.758
C09850=1080.062,77.872,434.984,174.123,21.995,153.758
C09851=1080.056,77.622,435.001,174.121,21.994,153.758
C09852=1080.050,77.373,435.019,174.119,21.991,153.758
C09853=1080.044,77.124,435.036,174.118,21.989,153.758
C09854=1080.039,76.875,435.053,174.116,21.987,153.757
C09855=1080.033,76.625,435.071,174.114,21.984,153.757
C09856=1080.027,76.376,435.088,174.113,21.982,153.757
C09857=1080.021,76.127,435.105,174.112,21.980,153.757
C09858=1080.016,75.877,435.122,174.109,21.977,153.757
C09859=1080.010,75.628,435.140,174.108,21.975,153.756
C09860=1080.003,75.379,435.157,174.106,21.972,153.756
C09861=1079.998,75.129,435.174,174.105,21.970,153.756
C09862=1079.993,74.880,435.191,174.103,21.968,153.756
C09863=1079.987,74.630,435.209,174.101,21.966,153.756
C09864=1079.981,74.381,435.226,174.100,21.963,153.755
C09865=1079.975,74.132,435.243,174.099,21.961,153.755
C09866=1079.970,73.883,435.260,174.097,21.959,153.755
C09867=1079.964,73.633,435.278,174.095,21.957,153.755
C09868=1079.958,73.383,435.294,174.093,21.954,153.754
C09869=1079.952,73.134,435.312,174.092,21.952,153.754
C09870=1079.947,72.885,435.329,174.091,21.949,153.754
C09871=1079.941,72.636,435.346,174.088,21.947,153.754
C09872=1079.935,72.387,435.363,174.087,21.945,153.753
C09873=1079.930,72.137,435.380,174.086,21.943,153.753
C09874=1079.923,71.888,435.397,174.084,21.940,153.753
C09875=1079.918,71.638,435.414,174.082,21.938,153.753
C09876=1079.913,71.389,435.432,174.081,21.935,153.753
C09877=1079.907,71.140,435.448,174.079,21.933,153.752
C09878=1079.901,70.891,435.466,174.078,21.931,153.752
C09879=1079.896,70.641,435.482,174.075,21.928,153.752
C09880=1079.889,70.392,435.500,174.074,21.926,153.752
C09881=1079.884,70.142,435.517,174.073,21.924,153.751
C09882=1079.878,69.893,435.534,174.071,21.921,153.751
C09883=1079.872,69.644,435.550,174.069,21.919,153.751
C09884=1079.867,69.394,435.567,174.068,21.917,153.751
C09885=1079.861,69.145,435.584,174.066,21.914,153.751
C09886=1079.856,68.896,435.601,174.065,21.912,153.750
C09887=1079.849,68.646,435.618,174.063,21.910,153.750
C09888=1079.844,68.397,435.635,174.061,21.907,153.750
C09889=1079.837,68.148,435.652,174.060,21.905,153.750
C09890=1079.832,67.898,435.669,174.059,21.903,153.749
C09891=1079.826,67.649,435.685,174.057,21.900,153.749
C09892=1079.821,67.400,435.703,174.055,21.898,153.749
C09893=1079.815,67.150,435.720,174.054,21.896,153.749
C09894=1079.810,66.901,435.736,174.052,21.893,153.749
C09895=1079.803,66.651,435.754,174.051,21.891,153.748
C09896=1079.797,66.402,435.770,174.048,21.888,153.748
C09897=1079.791,66.152,435.786,174.047,21.886,153.748
C09898=1079.786,65.903,435.804,174.046,21.884,153.748
C09899=1079.780,65.654,435.820,174.044,21.882,153.748
C09900=1079.775,65.404,435.837,174.043,21.879,153.747
C09901=1079.769,65.156,435.854,174.041,21.877,153.747
C09902=1079.763,64.906,435.871,174.039,21.874,153.747
C09903=1079.757,64.657,435.887,174.038,21.872,153.746
C09904=1079.752,64.407,435.905,174.037,21.870,153.746
C09905=1079.745,64.157,435.921,174.034,21.867,153.746
C09906=1079.739,63.908,435.938,174.033,21.865,153.746
C09907=1079.734,63.658,435.955,174.032,21.863,153.746
C09908=1079.727,63.379,435.973,174.030,21.860,153.745
C09909=1079.721,63.099,435.992,174.028,21.857,153.745
C09910=1079.715,62.819,436.010,174.026,21.855,153.745
C09911=1079.707,62.539,436.029,174.024,21.853,153.745
C09912=1079.702,62.289,436.046,174.023,21.850,153.744
C09913=1079.696,62.039,436.062,174.022,21.848,153.744
C09914=1079.689,61.791,436.079,174.020,21.845,153.744
C09915=1079.684,61.541,436.096,174.018,21.843,153.744
C09916=1079.678,61.292,436.112,174.017,21.841,153.744
C09917=1079.672,61.042,436.129,174.015,21.839,153.743
C09918=1079.666,60.793,436.145,174.014,21.836,153.743
C09919=1079.660,60.543,436.161,174.012,21.834,153.743
C09920=1079.655,60.294,436.179,174.010,21.831,153.743
C09921=1079.649,60.045,436.195,174.009,21.829,153.743
C09922=1079.643,59.796,436.211,174.008,21.827,153.742
C09923=1079.637,59.546,436.228,174.005,21.825,153.742
C09924=1079.632,59.297,436.244,174.004,21.822,153.742
C09925=1079.626,59.047,436.261,174.003,21.820,153.742
C09926=1079.620,58.798,436.277,174.001,21.817,153.741
C09927=1079.613,58.548,436.294,173.999,21.815,153.741
C09928=1079.608,58.298,436.310,173.998,21.813,153.741
C09929=1079.602,58.049,436.327,173.996,21.811,153.741
C09930=1079.596,57.800,436.344,173.995,21.808,153.740
C09931=1079.590,57.551,436.360,173.993,21.806,153.740
C09932=1079.584,57.302,436.376,173.991,21.803,153.740
C09933=1079.579,57.052,436.393,173.990,21.801,153.740
C09934=1079.573,56.803,436.409,173.989,21.799,153.740
C09935=1079.567,56.553,436.426,173.987,21.797,153.739
C09936=1079.561,56.304,436.442,173.985,21.794,153.739
C09937=1079.555,56.054,436.458,173.984,21.792,153.739
C09938=1079.550,55.805,436.475,173.982,21.789,153.739
C09939=1079.544,55.555,436.491,173.981,21.787,153.738
C09940=1079.539,55.307,436.507,173.979,21.785,153.738
C09941=1079.533,55.058,436.523,173.977,21.782,153.738
C09942=1079.527,54.808,436.540,173.976,21.780,153.738
C09943=1079.521,54.558,436.556,173.975,21.778,153.738
C09944=1079.516,54.309,436.572,173.974,21.776,153.737
C09945=1079.510,54.059,436.588,173.971,21.773,153.737
C09946=1079.504,53.810,436.604,173.970,21.770,153.737
C09947=1079.498,53.560,436.621,173.969,21.768,153.737
C09948=1079.492,53.311,436.637,173.967,21.766,153.736
C09949=1079.487,53.061,436.654,173.966,21.764,153.736
C09950=1079.481,52.812,436.670,173.964,21.761,153.736
C09951=1079.475,52.563,436.686,173.962,21.758,153.736
C09952=1079.469,52.313,436.703,173.961,21.756,153.735
C09953=1079.463,52.064,436.719,173.960,21.754,153.735
C09954=1079.457,51.815,436.735,173.958,21.752,153.735
C09955=1079.452,51.565,436.750,173.956,21.749,153.735
C09956=1079.447,51.316,436.767,173.955,21.747,153.734
C09957=1079.441,51.066,436.783,173.954,21.745,153.734
C09958=1079.435,50.817,436.800,173.952,21.742,153.734
C09959=1079.429,50.568,436.816,173.950,21.740,153.734
C09960=1079.423,50.318,436.832,173.949,21.737,153.734
C09961=1079.417,50.068,436.848,173.947,21.734,153.733
C09962=1079.411,49.819,436.864,173.946,21.733,153.733
C09963=1079.406,49.570,436.880,173.945,21.730,153.733
C09964=1079.401,49.321,436.897,173.943,21.727,153.733
C09965=1079.395,49.071,436.912,173.941,21.725,153.732
C09966=1079.389,48.821,436.928,173.940,21.723,153.732
C09967=1079.383,48.572,436.945,173.938,21.720,153.732
C09968=1079.377,48.323,436.961,173.937,21.718,153.732
C09969=1079.372,48.074,436.977,173.936,21.716,153.731
C09970=1079.366,47.824,436.992,173.934,21.714,153.731
C09971=1079.360,47.575,437.009,173.932,21.711,153.731
C09972=1079.354,47.294,437.027,173.931,21.708,153.731
C09973=1079.348,47.014,437.045,173.929,21.705,153.730
C09974=1079.341,46.734,437.063,173.928,21.703,153.730
C09975=1079.335,46.453,437.081,173.926,21.700,153.730
C09976=1079.329,46.204,437.096,173.925,21.698,153.729
C09977=1079.323,45.954,437.113,173.922,21.695,153.729
C09978=1079.318,45.706,437.129,173.921,21.693,153.729
C09979=1079.312,45.456,437.144,173.920,21.690,153.729
C09980=1079.307,45.206,437.161,173.918,21.688,153.729
C09981=1079.301,44.957,437.177,173.917,21.685,153.728
C09982=1079.296,44.707,437.192,173.915,21.683,153.728
C09983=1079.290,44.458,437.209,173.914,21.681,153.728
C09984=1079.284,44.209,437.225,173.912,21.678,153.728
C09985=1079.278,43.959,437.240,173.911,21.676,153.727
C09986=1079.273,43.710,437.256,173.909,21.674,153.727
C09987=1079.267,43.460,437.272,173.907,21.671,153.727
C09988=1079.261,43.211,437.288,173.906,21.668,153.727
C09989=1079.255,42.962,437.304,173.905,21.666,153.726
C09990=1079.249,42.712,437.319,173.904,21.664,153.726
C09991=1079.244,42.463,437.335,173.902,21.661,153.726
C09992=1079.238,42.213,437.351,173.900,21.659,153.726
C09993=1079.232,41.964,437.367,173.899,21.657,153.725
C09994=1079.226,41.714,437.383,173.897,21.654,153.725
C09995=1079.220,41.464,437.399,173.896,21.652,153.725
C09996=1079.215,41.215,437.413,173.895,21.649,153.725
//INST
///DATE 2021/06/25 14:45
///ATTR SC,RW,RJ
////FRAME ROBOT
///GROUP1 RB1
NOP
MOVL C00000 V=800.0 PL=0
MOVL C00001 V=800.0 PL=0
MOVL C00002 V=800.0 PL=0
MOVL C00003 V=800.0 PL=0
MOVL C00004 V=800.0 PL=0
MOVL C00005 V=800.0 PL=0
MOVL C00006 V=800.0 PL=0
MOVL C00007 V=800.0 PL=0
MOVL C00008 V=800.0 PL=0
MOVL C00009 V=800.0 PL=0
MOVL C00010 V=800.0 PL=0
MOVL C00011 V=800.0 PL=0
MOVL C00012 V=800.0 PL=0
MOVL C00013 V=800.0 PL=0
MOVL C00014 V=800.0 PL=0
MOVL C00015 V=800.0 PL=0
MOVL C00016 V=800.0 PL=0
MOVL C00017 V=800.0 PL=0
MOVL C00018 V=800.0 PL=0
MOVL C00019 V=800.0 PL=0
MOVL C00020 V=800.0 PL=0
MOVL C00021 V=800.0 PL=0
MOVL C00022 V=800.0 PL=0
MOVL C00023 V=800.0 PL=0
MOVL C00024 V=800.0 PL=0
MOVL C00025 V=800.0 PL=0
MOVL C00026 V=800.0 PL=0
MOVL C00027 V=800.0 PL=0
MOVL C00028 V=800.0 PL=0
MOVL C00029 V=800.0 PL=0
MOVL C00030 V=800.0 PL=0
MOVL C00031 V=800.0 PL=0
MOVL C00032 V=800.0 PL=0
MOVL C00033 V=800.0 PL=0
MOVL C00034 V=800.0 PL=0
MOVL C00035 V=800.0 PL=0
MOVL C00036 V=800.0 PL=0
MOVL C00037 V=800.0 PL=0
MOVL C00038 V=800.0 PL=0
MOVL C00039 V=800.0 PL=0
MOVL C00040 V=800.0 PL=0
MOVL C00041 V=800.0 PL=0
MOVL C00042 V=800.0 PL=0
MOVL C00043 V=800.0 PL=0
MOVL C00044 V=800.0 PL=0
MOVL C00045 V=800.0 PL=0
MOVL C00046 V=800.0 PL=0
MOVL C00047 V=800.0 PL=0
MOVL C00048 V=800.0 PL=0
MOVL C00049 V=800.0 PL=0
MOVL C00050 V=800.0 PL=0
MOVL C00051 V=800.0 PL=0
MOVL C00052 V=800.0 PL=0
MOVL C00053 V=800.0 PL=0
MOVL C00054 V=800.0 PL=0
MOVL C00055 V=800.0 PL=0
MOVL C00056 V=800.0 PL=0
MOVL C00057 V=800.0 PL=0
MOVL C00058 V=800.0 PL=0
MOVL C00059 V=800.0 PL=0
MOVL C00060 V=800.0 PL=0
MOVL C00061 V=800.0 PL=0
MOVL C00062 V=800.0 PL=0
MOVL C00063 V=800.0 PL=0
MOVL C00064 V=800.0 PL=0
MOVL C00065 V=800.0 PL=0
MOVL C00066 V=800.0 PL=0
MOVL C00067 V=800.0 PL=0
MOVL C00068 V=800.0 PL=0
MOVL C00069 V=800.0 PL=0
MOVL C00070 V=800.0 PL=0
MOVL C00071 V=800.0 PL=0
MOVL C00072 V=800.0 PL=0
MOVL C00073 V=800.0 PL=0
MOVL C00074 V=800.0 PL=0
MOVL C00075 V=800.0 PL=0
MOVL C00076 V=800.0 PL=0
MOVL C00077 V=800.0 PL=0
MOVL C00078 V=800.0 PL=0
MOVL C00079 V=800.0 PL=0
MOVL C00080 V=800.0 PL=0
MOVL C00081 V=800.0 PL=0
MOVL C00082 V=800.0 PL=0
MOVL C00083 V=800.0 PL=0
MOVL C00084 V=800.0 PL=0
MOVL C00085 V=800.0 PL=0
MOVL C00086 V=800.0 PL=0
MOVL C00087 V=800.0 PL=0
MOVL C00088 V=800.0 PL=0
MOVL C00089 V=800.0 PL=0
MOVL C00090 V=800.0 PL=0
MOVL C00091 V=800.0 PL=0
MOVL C00092 V=800.0 PL=0
MOVL C00093 V=800.0 PL=0
MOVL C00094 V=800.0 PL=0
MOVL C00095 V=800.0 PL=0
MOVL C00096 V=800.0 PL=0
MOVL C00097 V=800.0 PL=0
MOVL C00098 V=800.0 PL=0
MOVL C00099 V=800.0 PL=0
MOVL C00100 V=800.0 PL=0
MOVL C00101 V=800.0 PL=0
MOVL C00102 V=800.0 PL=0
MOVL C00103 V=800.0 PL=0
MOVL C00104 V=800.0 PL=0
MOVL C00105 V=800.0 PL=0
MOVL C00106 V=800.0 PL=0
MOVL C00107 V=800.0 PL=0
MOVL C00108 V=800.0 PL=0
MOVL C00109 V=800.0 PL=0
MOVL C00110 V=800.0 PL=0
MOVL C00111 V=800.0 PL=0
MOVL C00112 V=800.0 PL=0
MOVL C00113 V=800.0 PL=0
MOVL C00114 V=800.0 PL=0
MOVL C00115 V=800.0 PL=0
MOVL C00116 V=800.0 PL=0
MOVL C00117 V=800.0 PL=0
MOVL C00118 V=800.0 PL=0
MOVL C00119 V=800.0 PL=0
MOVL C00120 V=800.0 PL=0
MOVL C00121 V=800.0 PL=0
MOVL C00122 V=800.0 PL=0
MOVL C00123 V=800.0 PL=0
MOVL C00124 V=800.0 PL=0
MOVL C00125 V=800.0 PL=0
MOVL C00126 V=800.0 PL=0
MOVL C00127 V=800.0 PL=0
MOVL C00128 V=800.0 PL=0
MOVL C00129 V=800.0 PL=0
MOVL C00130 V=800.0 PL=0
MOVL C00131 V=800.0 PL=0
MOVL C00132 V=800.0 PL=0
MOVL C00133 V=800.0 PL=0
MOVL C00134 V=800.0 PL=0
MOVL C00135 V=800.0 PL=0
MOVL C00136 V=800.0 PL=0
MOVL C00137 V=800.0 PL=0
MOVL C00138 V=800.0 PL=0
MOVL C00139 V=800.0 PL=0
MOVL C00140 V=800.0 PL=0
MOVL C00141 V=800.0 PL=0
MOVL C00142 V=800.0 PL=0
MOVL C00143 V=800.0 PL=0
MOVL C00144 V=800.0 PL=0
MOVL C00145 V=800.0 PL=0
MOVL C00146 V=800.0 PL=0
MOVL C00147 V=800.0 PL=0
MOVL C00148 V=800.0 PL=0
MOVL C00149 V=800.0 PL=0
MOVL C00150 V=800.0 PL=0
MOVL C00151 V=800.0 PL=0
MOVL C00152 V=800.0 PL=0
MOVL C00153 V=800.0 PL=0
MOVL C00154 V=800.0 PL=0
MOVL C00155 V=800.0 PL=0
MOVL C00156 V=800.0 PL=0
MOVL C00157 V=800.0 PL=0
MOVL C00158 V=800.0 PL=0
MOVL C00159 V=800.0 PL=0
MOVL C00160 V=800.0 PL=0
MOVL C00161 V=800.0 PL=0
MOVL C00162 V=800.0 PL=0
MOVL C00163 V=800.0 PL=0
MOVL C00164 V=800.0 PL=0
MOVL C00165 V=800.0 PL=0
MOVL C00166 V=800.0 PL=0
MOVL C00167 V=800.0 PL=0
MOVL C00168 V=800.0 PL=0
MOVL C00169 V=800.0 PL=0
MOVL C00170 V=800.0 PL=0
MOVL C00171 V=800.0 PL=0
MOVL C00172 V=800.0 PL=0
MOVL C00173 V=800.0 PL=0
MOVL C00174 V=800.0 PL=0
MOVL C00175 V=800.0 PL=0
MOVL C00176 V=800.0 PL=0
MOVL C00177 V=800.0 PL=0
MOVL C00178 V=800.0 PL=0
MOVL C00179 V=800.0 PL=0
MOVL C00180 V=800.0 PL=0
MOVL C00181 V=800.0 PL=0
MOVL C00182 V=800.0 PL=0
MOVL C00183 V=800.0 PL=0
MOVL C00184 V=800.0 PL=0
MOVL C00185 V=800.0 PL=0
MOVL C00186 V=800.0 PL=0
MOVL C00187 V=800.0 PL=0
MOVL C00188 V=800.0 PL=0
MOVL C00189 V=800.0 PL=0
MOVL C00190 V=800.0 PL=0
MOVL C00191 V=800.0 PL=0
MOVL C00192 V=800.0 PL=0
MOVL C00193 V=800.0 PL=0
MOVL C00194 V=800.0 PL=0
MOVL C00195 V=800.0 PL=0
MOVL C00196 V=800.0 PL=0
MOVL C00197 V=800.0 PL=0
MOVL C00198 V=800.0 PL=0
MOVL C00199 V=800.0 PL=0
MOVL C00200 V=800.0 PL=0
MOVL C00201 V=800.0 PL=0
MOVL C00202 V=800.0 PL=0
MOVL C00203 V=800.0 PL=0
MOVL C00204 V=800.0 PL=0
MOVL C00205 V=800.0 PL=0
MOVL C00206 V=800.0 PL=0
MOVL C00207 V=800.0 PL=0
MOVL C00208 V=800.0 PL=0
MOVL C00209 V=800.0 PL=0
MOVL C00210 V=800.0 PL=0
MOVL C00211 V=800.0 PL=0
MOVL C00212 V=800.0 PL=0
MOVL C00213 V=800.0 PL=0
MOVL C00214 V=800.0 PL=0
MOVL C00215 V=800.0 PL=0
MOVL C00216 V=800.0 PL=0
MOVL C00217 V=800.0 PL=0
MOVL C00218 V=800.0 PL=0
MOVL C00219 V=800.0 PL=0
MOVL C00220 V=800.0 PL=0
MOVL C00221 V=800.0 PL=0
MOVL C00222 V=800.0 PL=0
MOVL C00223 V=800.0 PL=0
MOVL C00224 V=800.0 PL=0
MOVL C00225 V=800.0 PL=0
MOVL C00226 V=800.0 PL=0
MOVL C00227 V=800.0 PL=0
MOVL C00228 V=800.0 PL=0
MOVL C00229 V=800.0 PL=0
MOVL C00230 V=800.0 PL=0
MOVL C00231 V=800.0 PL=0
MOVL C00232 V=800.0 PL=0
MOVL C00233 V=800.0 PL=0
MOVL C00234 V=800.0 PL=0
MOVL C00235 V=800.0 PL=0
MOVL C00236 V=800.0 PL=0
MOVL C00237 V=800.0 PL=0
MOVL C00238 V=800.0 PL=0
MOVL C00239 V=800.0 PL=0
MOVL C00240 V=800.0 PL=0
MOVL C00241 V=800.0 PL=0
MOVL C00242 V=800.0 PL=0
MOVL C00243 V=800.0 PL=0
MOVL C00244 V=800.0 PL=0
MOVL C00245 V=800.0 PL=0
MOVL C00246 V=800.0 PL=0
MOVL C00247 V=800.0 PL=0
MOVL C00248 V=800.0 PL=0
MOVL C00249 V=800.0 PL=0
MOVL C00250 V=800.0 PL=0
MOVL C00251 V=800.0 PL=0
MOVL C00252 V=800.0 PL=0
MOVL C00253 V=800.0 PL=0
MOVL C00254 V=800.0 PL=0
MOVL C00255 V=800.0 PL=0
MOVL C00256 V=800.0 PL=0
MOVL C00257 V=800.0 PL=0
MOVL C00258 V=800.0 PL=0
MOVL C00259 V=800.0 PL=0
MOVL C00260 V=800.0 PL=0
MOVL C00261 V=800.0 PL=0
MOVL C00262 V=800.0 PL=0
MOVL C00263 V=800.0 PL=0
MOVL C00264 V=800.0 PL=0
MOVL C00265 V=800.0 PL=0
MOVL C00266 V=800.0 PL=0
MOVL C00267 V=800.0 PL=0
MOVL C00268 V=800.0 PL=0
MOVL C00269 V=800.0 PL=0
MOVL C00270 V=800.0 PL=0
MOVL C00271 V=800.0 PL=0
MOVL C00272 V=800.0 PL=0
MOVL C00273 V=800.0 PL=0
MOVL C00274 V=800.0 PL=0
MOVL C00275 V=800.0 PL=0
MOVL C00276 V=800.0 PL=0
MOVL C00277 V=800.0 PL=0
MOVL C00278 V=800.0 PL=0
MOVL C00279 V=800.0 PL=0
MOVL C00280 V=800.0 PL=0
MOVL C00281 V=800.0 PL=0
MOVL C00282 V=800.0 PL=0
MOVL C00283 V=800.0 PL=0
MOVL C00284 V=800.0 PL=0
MOVL C00285 V=800.0 PL=0
MOVL C00286 V=800.0 PL=0
MOVL C00287 V=800.0 PL=0
MOVL C00288 V=800.0 PL=0
MOVL C00289 V=800.0 PL=0
MOVL C00290 V=800.0 PL=0
MOVL C00291 V=800.0 PL=0
MOVL C00292 V=800.0 PL=0
MOVL C00293 V=800.0 PL=0
MOVL C00294 V=800.0 PL=0
MOVL C00295 V=800.0 PL=0
MOVL C00296 V=800.0 PL=0
MOVL C00297 V=800.0 PL=0
MOVL C00298 V=800.0 PL=0
MOVL C00299 V=800.0 PL=0
MOVL C00300 V=800.0 PL=0
MOVL C00301 V=800.0 PL=0
MOVL C00302 V=800.0 PL=0
MOVL C00303 V=800.0 PL=0
MOVL C00304 V=800.0 PL=0
MOVL C00305 V=800.0 PL=0
MOVL C00306 V=800.0 PL=0
MOVL C00307 V=800.0 PL=0
MOVL C00308 V=800.0 PL=0
MOVL C00309 V=800.0 PL=0
MOVL C00310 V=800.0 PL=0
MOVL C00311 V=800.0 PL=0
MOVL C00312 V=800.0 PL=0
MOVL C00313 V=800.0 PL=0
MOVL C00314 V=800.0 PL=0
MOVL C00315 V=800.0 PL=0
MOVL C00316 V=800.0 PL=0
MOVL C00317 V=800.0 PL=0
MOVL C00318 V=800.0 PL=0
MOVL C00319 V=800.0 PL=0
MOVL C00320 V=800.0 PL=0
MOVL C00321 V=800.0 PL=0
MOVL C00322 V=800.0 PL=0
MOVL C00323 V=800.0 PL=0
MOVL C00324 V=800.0 PL=0
MOVL C00325 V=800.0 PL=0
MOVL C00326 V=800.0 PL=0
MOVL C00327 V=800.0 PL=0
MOVL C00328 V=800.0 PL=0
MOVL C00329 V=800.0 PL=0
MOVL C00330 V=800.0 PL=0
MOVL C00331 V=800.0 PL=0
MOVL C00332 V=800.0 PL=0
MOVL C00333 V=800.0 PL=0
MOVL C00334 V=800.0 PL=0
MOVL C00335 V=800.0 PL=0
MOVL C00336 V=800.0 PL=0
MOVL C00337 V=800.0 PL=0
MOVL C00338 V=800.0 PL=0
MOVL C00339 V=800.0 PL=0
MOVL C00340 V=800.0 PL=0
MOVL C00341 V=800.0 PL=0
MOVL C00342 V=800.0 PL=0
MOVL C00343 V=800.0 PL=0
MOVL C00344 V=800.0 PL=0
MOVL C00345 V=800.0 PL=0
MOVL C00346 V=800.0 PL=0
MOVL C00347 V=800.0 PL=0
MOVL C00348 V=800.0 PL=0
MOVL C00349 V=800.0 PL=0
MOVL C00350 V=800.0 PL=0
MOVL C00351 V=800.0 PL=0
MOVL C00352 V=800.0 PL=0
MOVL C00353 V=800.0 PL=0
MOVL C00354 V=800.0 PL=0
MOVL C00355 V=800.0 PL=0
MOVL C00356 V=800.0 PL=0
MOVL C00357 V=800.0 PL=0
MOVL C00358 V=800.0 PL=0
MOVL C00359 V=800.0 PL=0
MOVL C00360 V=800.0 PL=0
MOVL C00361 V=800.0 PL=0
MOVL C00362 V=800.0 PL=0
MOVL C00363 V=800.0 PL=0
MOVL C00364 V=800.0 PL=0
MOVL C00365 V=800.0 PL=0
MOVL C00366 V=800.0 PL=0
MOVL C00367 V=800.0 PL=0
MOVL C00368 V=800.0 PL=0
MOVL C00369 V=800.0 PL=0
MOVL C00370 V=800.0 PL=0
MOVL C00371 V=800.0 PL=0
MOVL C00372 V=800.0 PL=0
MOVL C00373 V=800.0 PL=0
MOVL C00374 V=800.0 PL=0
MOVL C00375 V=800.0 PL=0
MOVL C00376 V=800.0 PL=0
MOVL C00377 V=800.0 PL=0
MOVL C00378 V=800.0 PL=0
MOVL C00379 V=800.0 PL=0
MOVL C00380 V=800.0 PL=0
MOVL C00381 V=800.0 PL=0
MOVL C00382 V=800.0 PL=0
MOVL C00383 V=800.0 PL=0
MOVL C00384 V=800.0 PL=0
MOVL C00385 V=800.0 PL=0
MOVL C00386 V=800.0 PL=0
MOVL C00387 V=800.0 PL=0
MOVL C00388 V=800.0 PL=0
MOVL C00389 V=800.0 PL=0
MOVL C00390 V=800.0 PL=0
MOVL C00391 V=800.0 PL=0
MOVL C00392 V=800.0 PL=0
MOVL C00393 V=800.0 PL=0
MOVL C00394 V=800.0 PL=0
MOVL C00395 V=800.0 PL=0
MOVL C00396 V=800.0 PL=0
MOVL C00397 V=800.0 PL=0
MOVL C00398 V=800.0 PL=0
MOVL C00399 V=800.0 PL=0
MOVL C00400 V=800.0 PL=0
MOVL C00401 V=800.0 PL=0
MOVL C00402 V=800.0 PL=0
MOVL C00403 V=800.0 PL=0
MOVL C00404 V=800.0 PL=0
MOVL C00405 V=800.0 PL=0
MOVL C00406 V=800.0 PL=0
MOVL C00407 V=800.0 PL=0
MOVL C00408 V=800.0 PL=0
MOVL C00409 V=800.0 PL=0
MOVL C00410 V=800.0 PL=0
MOVL C00411 V=800.0 PL=0
MOVL C00412 V=800.0 PL=0
MOVL C00413 V=800.0 PL=0
MOVL C00414 V=800.0 PL=0
MOVL C00415 V=800.0 PL=0
MOVL C00416 V=800.0 PL=0
MOVL C00417 V=800.0 PL=0
MOVL C00418 V=800.0 PL=0
MOVL C00419 V=800.0 PL=0
MOVL C00420 V=800.0 PL=0
MOVL C00421 V=800.0 PL=0
MOVL C00422 V=800.0 PL=0
MOVL C00423 V=800.0 PL=0
MOVL C00424 V=800.0 PL=0
MOVL C00425 V=800.0 PL=0
MOVL C00426 V=800.0 PL=0
MOVL C00427 V=800.0 PL=0
MOVL C00428 V=800.0 PL=0
MOVL C00429 V=800.0 PL=0
MOVL C00430 V=800.0 PL=0
MOVL C00431 V=800.0 PL=0
MOVL C00432 V=800.0 PL=0
MOVL C00433 V=800.0 PL=0
MOVL C00434 V=800.0 PL=0
MOVL C00435 V=800.0 PL=0
MOVL C00436 V=800.0 PL=0
MOVL C00437 V=800.0 PL=0
MOVL C00438 V=800.0 PL=0
MOVL C00439 V=800.0 PL=0
MOVL C00440 V=800.0 PL=0
MOVL C00441 V=800.0 PL=0
MOVL C00442 V=800.0 PL=0
MOVL C00443 V=800.0 PL=0
MOVL C00444 V=800.0 PL=0
MOVL C00445 V=800.0 PL=0
MOVL C00446 V=800.0 PL=0
MOVL C00447 V=800.0 PL=0
MOVL C00448 V=800.0 PL=0
MOVL C00449 V=800.0 PL=0
MOVL C00450 V=800.0 PL=0
MOVL C00451 V=800.0 PL=0
MOVL C00452 V=800.0 PL=0
MOVL C00453 V=800.0 PL=0
MOVL C00454 V=800.0 PL=0
MOVL C00455 V=800.0 PL=0
MOVL C00456 V=800.0 PL=0
MOVL C00457 V=800.0 PL=0
MOVL C00458 V=800.0 PL=0
MOVL C00459 V=800.0 PL=0
MOVL C00460 V=800.0 PL=0
MOVL C00461 V=800.0 PL=0
MOVL C00462 V=800.0 PL=0
MOVL C00463 V=800.0 PL=0
MOVL C00464 V=800.0 PL=0
MOVL C00465 V=800.0 PL=0
MOVL C00466 V=800.0 PL=0
MOVL C00467 V=800.0 PL=0
MOVL C00468 V=800.0 PL=0
MOVL C00469 V=800.0 PL=0
MOVL C00470 V=800.0 PL=0
MOVL C00471 V=800.0 PL=0
MOVL C00472 V=800.0 PL=0
MOVL C00473 V=800.0 PL=0
MOVL C00474 V=800.0 PL=0
MOVL C00475 V=800.0 PL=0
MOVL C00476 V=800.0 PL=0
MOVL C00477 V=800.0 PL=0
MOVL C00478 V=800.0 PL=0
MOVL C00479 V=800.0 PL=0
MOVL C00480 V=800.0 PL=0
MOVL C00481 V=800.0 PL=0
MOVL C00482 V=800.0 PL=0
MOVL C00483 V=800.0 PL=0
MOVL C00484 V=800.0 PL=0
MOVL C00485 V=800.0 PL=0
MOVL C00486 V=800.0 PL=0
MOVL C00487 V=800.0 PL=0
MOVL C00488 V=800.0 PL=0
MOVL C00489 V=800.0 PL=0
MOVL C00490 V=800.0 PL=0
MOVL C00491 V=800.0 PL=0
MOVL C00492 V=800.0 PL=0
MOVL C00493 V=800.0 PL=0
MOVL C00494 V=800.0 PL=0
MOVL C00495 V=800.0 PL=0
MOVL C00496 V=800.0 PL=0
MOVL C00497 V=800.0 PL=0
MOVL C00498 V=800.0 PL=0
MOVL C00499 V=800.0 PL=0
MOVL C00500 V=800.0 PL=0
MOVL C00501 V=800.0 PL=0
MOVL C00502 V=800.0 PL=0
MOVL C00503 V=800.0 PL=0
MOVL C00504 V=800.0 PL=0
MOVL C00505 V=800.0 PL=0
MOVL C00506 V=800.0 PL=0
MOVL C00507 V=800.0 PL=0
MOVL C00508 V=800.0 PL=0
MOVL C00509 V=800.0 PL=0
MOVL C00510 V=800.0 PL=0
MOVL C00511 V=800.0 PL=0
MOVL C00512 V=800.0 PL=0
MOVL C00513 V=800.0 PL=0
MOVL C00514 V=800.0 PL=0
MOVL C00515 V=800.0 PL=0
MOVL C00516 V=800.0 PL=0
MOVL C00517 V=800.0 PL=0
MOVL C00518 V=800.0 PL=0
MOVL C00519 V=800.0 PL=0
MOVL C00520 V=800.0 PL=0
MOVL C00521 V=800.0 PL=0
MOVL C00522 V=800.0 PL=0
MOVL C00523 V=800.0 PL=0
MOVL C00524 V=800.0 PL=0
MOVL C00525 V=800.0 PL=0
MOVL C00526 V=800.0 PL=0
MOVL C00527 V=800.0 PL=0
MOVL C00528 V=800.0 PL=0
MOVL C00529 V=800.0 PL=0
MOVL C00530 V=800.0 PL=0
MOVL C00531 V=800.0 PL=0
MOVL C00532 V=800.0 PL=0
MOVL C00533 V=800.0 PL=0
MOVL C00534 V=800.0 PL=0
MOVL C00535 V=800.0 PL=0
MOVL C00536 V=800.0 PL=0
MOVL C00537 V=800.0 PL=0
MOVL C00538 V=800.0 PL=0
MOVL C00539 V=800.0 PL=0
MOVL C00540 V=800.0 PL=0
MOVL C00541 V=800.0 PL=0
MOVL C00542 V=800.0 PL=0
MOVL C00543 V=800.0 PL=0
MOVL C00544 V=800.0 PL=0
MOVL C00545 V=800.0 PL=0
MOVL C00546 V=800.0 PL=0
MOVL C00547 V=800.0 PL=0
MOVL C00548 V=800.0 PL=0
MOVL C00549 V=800.0 PL=0
MOVL C00550 V=800.0 PL=0
MOVL C00551 V=800.0 PL=0
MOVL C00552 V=800.0 PL=0
MOVL C00553 V=800.0 PL=0
MOVL C00554 V=800.0 PL=0
MOVL C00555 V=800.0 PL=0
MOVL C00556 V=800.0 PL=0
MOVL C00557 V=800.0 PL=0
MOVL C00558 V=800.0 PL=0
MOVL C00559 V=800.0 PL=0
MOVL C00560 V=800.0 PL=0
MOVL C00561 V=800.0 PL=0
MOVL C00562 V=800.0 PL=0
MOVL C00563 V=800.0 PL=0
MOVL C00564 V=800.0 PL=0
MOVL C00565 V=800.0 PL=0
MOVL C00566 V=800.0 PL=0
MOVL C00567 V=800.0 PL=0
MOVL C00568 V=800.0 PL=0
MOVL C00569 V=800.0 PL=0
MOVL C00570 V=800.0 PL=0
MOVL C00571 V=800.0 PL=0
MOVL C00572 V=800.0 PL=0
MOVL C00573 V=800.0 PL=0
MOVL C00574 V=800.0 PL=0
MOVL C00575 V=800.0 PL=0
MOVL C00576 V=800.0 PL=0
MOVL C00577 V=800.0 PL=0
MOVL C00578 V=800.0 PL=0
MOVL C00579 V=800.0 PL=0
MOVL C00580 V=800.0 PL=0
MOVL C00581 V=800.0 PL=0
MOVL C00582 V=800.0 PL=0
MOVL C00583 V=800.0 PL=0
MOVL C00584 V=800.0 PL=0
MOVL C00585 V=800.0 PL=0
MOVL C00586 V=800.0 PL=0
MOVL C00587 V=800.0 PL=0
MOVL C00588 V=800.0 PL=0
MOVL C00589 V=800.0 PL=0
MOVL C00590 V=800.0 PL=0
MOVL C00591 V=800.0 PL=0
MOVL C00592 V=800.0 PL=0
MOVL C00593 V=800.0 PL=0
MOVL C00594 V=800.0 PL=0
MOVL C00595 V=800.0 PL=0
MOVL C00596 V=800.0 PL=0
MOVL C00597 V=800.0 PL=0
MOVL C00598 V=800.0 PL=0
MOVL C00599 V=800.0 PL=0
MOVL C00600 V=800.0 PL=0
MOVL C00601 V=800.0 PL=0
MOVL C00602 V=800.0 PL=0
MOVL C00603 V=800.0 PL=0
MOVL C00604 V=800.0 PL=0
MOVL C00605 V=800.0 PL=0
MOVL C00606 V=800.0 PL=0
MOVL C00607 V=800.0 PL=0
MOVL C00608 V=800.0 PL=0
MOVL C00609 V=800.0 PL=0
MOVL C00610 V=800.0 PL=0
MOVL C00611 V=800.0 PL=0
MOVL C00612 V=800.0 PL=0
MOVL C00613 V=800.0 PL=0
MOVL C00614 V=800.0 PL=0
MOVL C00615 V=800.0 PL=0
MOVL C00616 V=800.0 PL=0
MOVL C00617 V=800.0 PL=0
MOVL C00618 V=800.0 PL=0
MOVL C00619 V=800.0 PL=0
MOVL C00620 V=800.0 PL=0
MOVL C00621 V=800.0 PL=0
MOVL C00622 V=800.0 PL=0
MOVL C00623 V=800.0 PL=0
MOVL C00624 V=800.0 PL=0
MOVL C00625 V=800.0 PL=0
MOVL C00626 V=800.0 PL=0
MOVL C00627 V=800.0 PL=0
MOVL C00628 V=800.0 PL=0
MOVL C00629 V=800.0 PL=0
MOVL C00630 V=800.0 PL=0
MOVL C00631 V=800.0 PL=0
MOVL C00632 V=800.0 PL=0
MOVL C00633 V=800.0 PL=0
MOVL C00634 V=800.0 PL=0
MOVL C00635 V=800.0 PL=0
MOVL C00636 V=800.0 PL=0
MOVL C00637 V=800.0 PL=0
MOVL C00638 V=800.0 PL=0
MOVL C00639 V=800.0 PL=0
MOVL C00640 V=800.0 PL=0
MOVL C00641 V=800.0 PL=0
MOVL C00642 V=800.0 PL=0
MOVL C00643 V=800.0 PL=0
MOVL C00644 V=800.0 PL=0
MOVL C00645 V=800.0 PL=0
MOVL C00646 V=800.0 PL=0
MOVL C00647 V=800.0 PL=0
MOVL C00648 V=800.0 PL=0
MOVL C00649 V=800.0 PL=0
MOVL C00650 V=800.0 PL=0
MOVL C00651 V=800.0 PL=0
MOVL C00652 V=800.0 PL=0
MOVL C00653 V=800.0 PL=0
MOVL C00654 V=800.0 PL=0
MOVL C00655 V=800.0 PL=0
MOVL C00656 V=800.0 PL=0
MOVL C00657 V=800.0 PL=0
MOVL C00658 V=800.0 PL=0
MOVL C00659 V=800.0 PL=0
MOVL C00660 V=800.0 PL=0
MOVL C00661 V=800.0 PL=0
MOVL C00662 V=800.0 PL=0
MOVL C00663 V=800.0 PL=0
MOVL C00664 V=800.0 PL=0
MOVL C00665 V=800.0 PL=0
MOVL C00666 V=800.0 PL=0
MOVL C00667 V=800.0 PL=0
MOVL C00668 V=800.0 PL=0
MOVL C00669 V=800.0 PL=0
MOVL C00670 V=800.0 PL=0
MOVL C00671 V=800.0 PL=0
MOVL C00672 V=800.0 PL=0
MOVL C00673 V=800.0 PL=0
MOVL C00674 V=800.0 PL=0
MOVL C00675 V=800.0 PL=0
MOVL C00676 V=800.0 PL=0
MOVL C00677 V=800.0 PL=0
MOVL C00678 V=800.0 PL=0
MOVL C00679 V=800.0 PL=0
MOVL C00680 V=800.0 PL=0
MOVL C00681 V=800.0 PL=0
MOVL C00682 V=800.0 PL=0
MOVL C00683 V=800.0 PL=0
MOVL C00684 V=800.0 PL=0
MOVL C00685 V=800.0 PL=0
MOVL C00686 V=800.0 PL=0
MOVL C00687 V=800.0 PL=0
MOVL C00688 V=800.0 PL=0
MOVL C00689 V=800.0 PL=0
MOVL C00690 V=800.0 PL=0
MOVL C00691 V=800.0 PL=0
MOVL C00692 V=800.0 PL=0
MOVL C00693 V=800.0 PL=0
MOVL C00694 V=800.0 PL=0
MOVL C00695 V=800.0 PL=0
MOVL C00696 V=800.0 PL=0
MOVL C00697 V=800.0 PL=0
MOVL C00698 V=800.0 PL=0
MOVL C00699 V=800.0 PL=0
MOVL C00700 V=800.0 PL=0
MOVL C00701 V=800.0 PL=0
MOVL C00702 V=800.0 PL=0
MOVL C00703 V=800.0 PL=0
MOVL C00704 V=800.0 PL=0
MOVL C00705 V=800.0 PL=0
MOVL C00706 V=800.0 PL=0
MOVL C00707 V=800.0 PL=0
MOVL C00708 V=800.0 PL=0
MOVL C00709 V=800.0 PL=0
MOVL C00710 V=800.0 PL=0
MOVL C00711 V=800.0 PL=0
MOVL C00712 V=800.0 PL=0
MOVL C00713 V=800.0 PL=0
MOVL C00714 V=800.0 PL=0
MOVL C00715 V=800.0 PL=0
MOVL C00716 V=800.0 PL=0
MOVL C00717 V=800.0 PL=0
MOVL C00718 V=800.0 PL=0
MOVL C00719 V=800.0 PL=0
MOVL C00720 V=800.0 PL=0
MOVL C00721 V=800.0 PL=0
MOVL C00722 V=800.0 PL=0
MOVL C00723 V=800.0 PL=0
MOVL C00724 V=800.0 PL=0
MOVL C00725 V=800.0 PL=0
MOVL C00726 V=800.0 PL=0
MOVL C00727 V=800.0 PL=0
MOVL C00728 V=800.0 PL=0
MOVL C00729 V=800.0 PL=0
MOVL C00730 V=800.0 PL=0
MOVL C00731 V=800.0 PL=0
MOVL C00732 V=800.0 PL=0
MOVL C00733 V=800.0 PL=0
MOVL C00734 V=800.0 PL=0
MOVL C00735 V=800.0 PL=0
MOVL C00736 V=800.0 PL=0
MOVL C00737 V=800.0 PL=0
MOVL C00738 V=800.0 PL=0
MOVL C00739 V=800.0 PL=0
MOVL C00740 V=800.0 PL=0
MOVL C00741 V=800.0 PL=0
MOVL C00742 V=800.0 PL=0
MOVL C00743 V=800.0 PL=0
MOVL C00744 V=800.0 PL=0
MOVL C00745 V=800.0 PL=0
MOVL C00746 V=800.0 PL=0
MOVL C00747 V=800.0 PL=0
MOVL C00748 V=800.0 PL=0
MOVL C00749 V=800.0 PL=0
MOVL C00750 V=800.0 PL=0
MOVL C00751 V=800.0 PL=0
MOVL C00752 V=800.0 PL=0
MOVL C00753 V=800.0 PL=0
MOVL C00754 V=800.0 PL=0
MOVL C00755 V=800.0 PL=0
MOVL C00756 V=800.0 PL=0
MOVL C00757 V=800.0 PL=0
MOVL C00758 V=800.0 PL=0
MOVL C00759 V=800.0 PL=0
MOVL C00760 V=800.0 PL=0
MOVL C00761 V=800.0 PL=0
MOVL C00762 V=800.0 PL=0
MOVL C00763 V=800.0 PL=0
MOVL C00764 V=800.0 PL=0
MOVL C00765 V=800.0 PL=0
MOVL C00766 V=800.0 PL=0
MOVL C00767 V=800.0 PL=0
MOVL C00768 V=800.0 PL=0
MOVL C00769 V=800.0 PL=0
MOVL C00770 V=800.0 PL=0
MOVL C00771 V=800.0 PL=0
MOVL C00772 V=800.0 PL=0
MOVL C00773 V=800.0 PL=0
MOVL C00774 V=800.0 PL=0
MOVL C00775 V=800.0 PL=0
MOVL C00776 V=800.0 PL=0
MOVL C00777 V=800.0 PL=0
MOVL C00778 V=800.0 PL=0
MOVL C00779 V=800.0 PL=0
MOVL C00780 V=800.0 PL=0
MOVL C00781 V=800.0 PL=0
MOVL C00782 V=800.0 PL=0
MOVL C00783 V=800.0 PL=0
MOVL C00784 V=800.0 PL=0
MOVL C00785 V=800.0 PL=0
MOVL C00786 V=800.0 PL=0
MOVL C00787 V=800.0 PL=0
MOVL C00788 V=800.0 PL=0
MOVL C00789 V=800.0 PL=0
MOVL C00790 V=800.0 PL=0
MOVL C00791 V=800.0 PL=0
MOVL C00792 V=800.0 PL=0
MOVL C00793 V=800.0 PL=0
MOVL C00794 V=800.0 PL=0
MOVL C00795 V=800.0 PL=0
MOVL C00796 V=800.0 PL=0
MOVL C00797 V=800.0 PL=0
MOVL C00798 V=800.0 PL=0
MOVL C00799 V=800.0 PL=0
MOVL C00800 V=800.0 PL=0
MOVL C00801 V=800.0 PL=0
MOVL C00802 V=800.0 PL=0
MOVL C00803 V=800.0 PL=0
MOVL C00804 V=800.0 PL=0
MOVL C00805 V=800.0 PL=0
MOVL C00806 V=800.0 PL=0
MOVL C00807 V=800.0 PL=0
MOVL C00808 V=800.0 PL=0
MOVL C00809 V=800.0 PL=0
MOVL C00810 V=800.0 PL=0
MOVL C00811 V=800.0 PL=0
MOVL C00812 V=800.0 PL=0
MOVL C00813 V=800.0 PL=0
MOVL C00814 V=800.0 PL=0
MOVL C00815 V=800.0 PL=0
MOVL C00816 V=800.0 PL=0
MOVL C00817 V=800.0 PL=0
MOVL C00818 V=800.0 PL=0
MOVL C00819 V=800.0 PL=0
MOVL C00820 V=800.0 PL=0
MOVL C00821 V=800.0 PL=0
MOVL C00822 V=800.0 PL=0
MOVL C00823 V=800.0 PL=0
MOVL C00824 V=800.0 PL=0
MOVL C00825 V=800.0 PL=0
MOVL C00826 V=800.0 PL=0
MOVL C00827 V=800.0 PL=0
MOVL C00828 V=800.0 PL=0
MOVL C00829 V=800.0 PL=0
MOVL C00830 V=800.0 PL=0
MOVL C00831 V=800.0 PL=0
MOVL C00832 V=800.0 PL=0
MOVL C00833 V=800.0 PL=0
MOVL C00834 V=800.0 PL=0
MOVL C00835 V=800.0 PL=0
MOVL C00836 V=800.0 PL=0
MOVL C00837 V=800.0 PL=0
MOVL C00838 V=800.0 PL=0
MOVL C00839 V=800.0 PL=0
MOVL C00840 V=800.0 PL=0
MOVL C00841 V=800.0 PL=0
MOVL C00842 V=800.0 PL=0
MOVL C00843 V=800.0 PL=0
MOVL C00844 V=800.0 PL=0
MOVL C00845 V=800.0 PL=0
MOVL C00846 V=800.0 PL=0
MOVL C00847 V=800.0 PL=0
MOVL C00848 V=800.0 PL=0
MOVL C00849 V=800.0 PL=0
MOVL C00850 V=800.0 PL=0
MOVL C00851 V=800.0 PL=0
MOVL C00852 V=800.0 PL=0
MOVL C00853 V=800.0 PL=0
MOVL C00854 V=800.0 PL=0
MOVL C00855 V=800.0 PL=0
MOVL C00856 V=800.0 PL=0
MOVL C00857 V=800.0 PL=0
MOVL C00858 V=800.0 PL=0
MOVL C00859 V=800.0 PL=0
MOVL C00860 V=800.0 PL=0
MOVL C00861 V=800.0 PL=0
MOVL C00862 V=800.0 PL=0
MOVL C00863 V=800.0 PL=0
MOVL C00864 V=800.0 PL=0
MOVL C00865 V=800.0 PL=0
MOVL C00866 V=800.0 PL=0
MOVL C00867 V=800.0 PL=0
MOVL C00868 V=800.0 PL=0
MOVL C00869 V=800.0 PL=0
MOVL C00870 V=800.0 PL=0
MOVL C00871 V=800.0 PL=0
MOVL C00872 V=800.0 PL=0
MOVL C00873 V=800.0 PL=0
MOVL C00874 V=800.0 PL=0
MOVL C00875 V=800.0 PL=0
MOVL C00876 V=800.0 PL=0
MOVL C00877 V=800.0 PL=0
MOVL C00878 V=800.0 PL=0
MOVL C00879 V=800.0 PL=0
MOVL C00880 V=800.0 PL=0
MOVL C00881 V=800.0 PL=0
MOVL C00882 V=800.0 PL=0
MOVL C00883 V=800.0 PL=0
MOVL C00884 V=800.0 PL=0
MOVL C00885 V=800.0 PL=0
MOVL C00886 V=800.0 PL=0
MOVL C00887 V=800.0 PL=0
MOVL C00888 V=800.0 PL=0
MOVL C00889 V=800.0 PL=0
MOVL C00890 V=800.0 PL=0
MOVL C00891 V=800.0 PL=0
MOVL C00892 V=800.0 PL=0
MOVL C00893 V=800.0 PL=0
MOVL C00894 V=800.0 PL=0
MOVL C00895 V=800.0 PL=0
MOVL C00896 V=800.0 PL=0
MOVL C00897 V=800.0 PL=0
MOVL C00898 V=800.0 PL=0
MOVL C00899 V=800.0 PL=0
MOVL C00900 V=800.0 PL=0
MOVL C00901 V=800.0 PL=0
MOVL C00902 V=800.0 PL=0
MOVL C00903 V=800.0 PL=0
MOVL C00904 V=800.0 PL=0
MOVL C00905 V=800.0 PL=0
MOVL C00906 V=800.0 PL=0
MOVL C00907 V=800.0 PL=0
MOVL C00908 V=800.0 PL=0
MOVL C00909 V=800.0 PL=0
MOVL C00910 V=800.0 PL=0
MOVL C00911 V=800.0 PL=0
MOVL C00912 V=800.0 PL=0
MOVL C00913 V=800.0 PL=0
MOVL C00914 V=800.0 PL=0
MOVL C00915 V=800.0 PL=0
MOVL C00916 V=800.0 PL=0
MOVL C00917 V=800.0 PL=0
MOVL C00918 V=800.0 PL=0
MOVL C00919 V=800.0 PL=0
MOVL C00920 V=800.0 PL=0
MOVL C00921 V=800.0 PL=0
MOVL C00922 V=800.0 PL=0
MOVL C00923 V=800.0 PL=0
MOVL C00924 V=800.0 PL=0
MOVL C00925 V=800.0 PL=0
MOVL C00926 V=800.0 PL=0
MOVL C00927 V=800.0 PL=0
MOVL C00928 V=800.0 PL=0
MOVL C00929 V=800.0 PL=0
MOVL C00930 V=800.0 PL=0
MOVL C00931 V=800.0 PL=0
MOVL C00932 V=800.0 PL=0
MOVL C00933 V=800.0 PL=0
MOVL C00934 V=800.0 PL=0
MOVL C00935 V=800.0 PL=0
MOVL C00936 V=800.0 PL=0
MOVL C00937 V=800.0 PL=0
MOVL C00938 V=800.0 PL=0
MOVL C00939 V=800.0 PL=0
MOVL C00940 V=800.0 PL=0
MOVL C00941 V=800.0 PL=0
MOVL C00942 V=800.0 PL=0
MOVL C00943 V=800.0 PL=0
MOVL C00944 V=800.0 PL=0
MOVL C00945 V=800.0 PL=0
MOVL C00946 V=800.0 PL=0
MOVL C00947 V=800.0 PL=0
MOVL C00948 V=800.0 PL=0
MOVL C00949 V=800.0 PL=0
MOVL C00950 V=800.0 PL=0
MOVL C00951 V=800.0 PL=0
MOVL C00952 V=800.0 PL=0
MOVL C00953 V=800.0 PL=0
MOVL C00954 V=800.0 PL=0
MOVL C00955 V=800.0 PL=0
MOVL C00956 V=800.0 PL=0
MOVL C00957 V=800.0 PL=0
MOVL C00958 V=800.0 PL=0
MOVL C00959 V=800.0 PL=0
MOVL C00960 V=800.0 PL=0
MOVL C00961 V=800.0 PL=0
MOVL C00962 V=800.0 PL=0
MOVL C00963 V=800.0 PL=0
MOVL C00964 V=800.0 PL=0
MOVL C00965 V=800.0 PL=0
MOVL C00966 V=800.0 PL=0
MOVL C00967 V=800.0 PL=0
MOVL C00968 V=800.0 PL=0
MOVL C00969 V=800.0 PL=0
MOVL C00970 V=800.0 PL=0
MOVL C00971 V=800.0 PL=0
MOVL C00972 V=800.0 PL=0
MOVL C00973 V=800.0 PL=0
MOVL C00974 V=800.0 PL=0
MOVL C00975 V=800.0 PL=0
MOVL C00976 V=800.0 PL=0
MOVL C00977 V=800.0 PL=0
MOVL C00978 V=800.0 PL=0
MOVL C00979 V=800.0 PL=0
MOVL C00980 V=800.0 PL=0
MOVL C00981 V=800.0 PL=0
MOVL C00982 V=800.0 PL=0
MOVL C00983 V=800.0 PL=0
MOVL C00984 V=800.0 PL=0
MOVL C00985 V=800.0 PL=0
MOVL C00986 V=800.0 PL=0
MOVL C00987 V=800.0 PL=0
MOVL C00988 V=800.0 PL=0
MOVL C00989 V=800.0 PL=0
MOVL C00990 V=800.0 PL=0
MOVL C00991 V=800.0 PL=0
MOVL C00992 V=800.0 PL=0
MOVL C00993 V=800.0 PL=0
MOVL C00994 V=800.0 PL=0
MOVL C00995 V=800.0 PL=0
MOVL C00996 V=800.0 PL=0
MOVL C00997 V=800.0 PL=0
MOVL C00998 V=800.0 PL=0
MOVL C00999 V=800.0 PL=0
MOVL C01000 V=800.0 PL=0
MOVL C01001 V=800.0 PL=0
MOVL C01002 V=800.0 PL=0
MOVL C01003 V=800.0 PL=0
MOVL C01004 V=800.0 PL=0
MOVL C01005 V=800.0 PL=0
MOVL C01006 V=800.0 PL=0
MOVL C01007 V=800.0 PL=0
MOVL C01008 V=800.0 PL=0
MOVL C01009 V=800.0 PL=0
MOVL C01010 V=800.0 PL=0
MOVL C01011 V=800.0 PL=0
MOVL C01012 V=800.0 PL=0
MOVL C01013 V=800.0 PL=0
MOVL C01014 V=800.0 PL=0
MOVL C01015 V=800.0 PL=0
MOVL C01016 V=800.0 PL=0
MOVL C01017 V=800.0 PL=0
MOVL C01018 V=800.0 PL=0
MOVL C01019 V=800.0 PL=0
MOVL C01020 V=800.0 PL=0
MOVL C01021 V=800.0 PL=0
MOVL C01022 V=800.0 PL=0
MOVL C01023 V=800.0 PL=0
MOVL C01024 V=800.0 PL=0
MOVL C01025 V=800.0 PL=0
MOVL C01026 V=800.0 PL=0
MOVL C01027 V=800.0 PL=0
MOVL C01028 V=800.0 PL=0
MOVL C01029 V=800.0 PL=0
MOVL C01030 V=800.0 PL=0
MOVL C01031 V=800.0 PL=0
MOVL C01032 V=800.0 PL=0
MOVL C01033 V=800.0 PL=0
MOVL C01034 V=800.0 PL=0
MOVL C01035 V=800.0 PL=0
MOVL C01036 V=800.0 PL=0
MOVL C01037 V=800.0 PL=0
MOVL C01038 V=800.0 PL=0
MOVL C01039 V=800.0 PL=0
MOVL C01040 V=800.0 PL=0
MOVL C01041 V=800.0 PL=0
MOVL C01042 V=800.0 PL=0
MOVL C01043 V=800.0 PL=0
MOVL C01044 V=800.0 PL=0
MOVL C01045 V=800.0 PL=0
MOVL C01046 V=800.0 PL=0
MOVL C01047 V=800.0 PL=0
MOVL C01048 V=800.0 PL=0
MOVL C01049 V=800.0 PL=0
MOVL C01050 V=800.0 PL=0
MOVL C01051 V=800.0 PL=0
MOVL C01052 V=800.0 PL=0
MOVL C01053 V=800.0 PL=0
MOVL C01054 V=800.0 PL=0
MOVL C01055 V=800.0 PL=0
MOVL C01056 V=800.0 PL=0
MOVL C01057 V=800.0 PL=0
MOVL C01058 V=800.0 PL=0
MOVL C01059 V=800.0 PL=0
MOVL C01060 V=800.0 PL=0
MOVL C01061 V=800.0 PL=0
MOVL C01062 V=800.0 PL=0
MOVL C01063 V=800.0 PL=0
MOVL C01064 V=800.0 PL=0
MOVL C01065 V=800.0 PL=0
MOVL C01066 V=800.0 PL=0
MOVL C01067 V=800.0 PL=0
MOVL C01068 V=800.0 PL=0
MOVL C01069 V=800.0 PL=0
MOVL C01070 V=800.0 PL=0
MOVL C01071 V=800.0 PL=0
MOVL C01072 V=800.0 PL=0
MOVL C01073 V=800.0 PL=0
MOVL C01074 V=800.0 PL=0
MOVL C01075 V=800.0 PL=0
MOVL C01076 V=800.0 PL=0
MOVL C01077 V=800.0 PL=0
MOVL C01078 V=800.0 PL=0
MOVL C01079 V=800.0 PL=0
MOVL C01080 V=800.0 PL=0
MOVL C01081 V=800.0 PL=0
MOVL C01082 V=800.0 PL=0
MOVL C01083 V=800.0 PL=0
MOVL C01084 V=800.0 PL=0
MOVL C01085 V=800.0 PL=0
MOVL C01086 V=800.0 PL=0
MOVL C01087 V=800.0 PL=0
MOVL C01088 V=800.0 PL=0
MOVL C01089 V=800.0 PL=0
MOVL C01090 V=800.0 PL=0
MOVL C01091 V=800.0 PL=0
MOVL C01092 V=800.0 PL=0
MOVL C01093 V=800.0 PL=0
MOVL C01094 V=800.0 PL=0
MOVL C01095 V=800.0 PL=0
MOVL C01096 V=800.0 PL=0
MOVL C01097 V=800.0 PL=0
MOVL C01098 V=800.0 PL=0
MOVL C01099 V=800.0 PL=0
MOVL C01100 V=800.0 PL=0
MOVL C01101 V=800.0 PL=0
MOVL C01102 V=800.0 PL=0
MOVL C01103 V=800.0 PL=0
MOVL C01104 V=800.0 PL=0
MOVL C01105 V=800.0 PL=0
MOVL C01106 V=800.0 PL=0
MOVL C01107 V=800.0 PL=0
MOVL C01108 V=800.0 PL=0
MOVL C01109 V=800.0 PL=0
MOVL C01110 V=800.0 PL=0
MOVL C01111 V=800.0 PL=0
MOVL C01112 V=800.0 PL=0
MOVL C01113 V=800.0 PL=0
MOVL C01114 V=800.0 PL=0
MOVL C01115 V=800.0 PL=0
MOVL C01116 V=800.0 PL=0
MOVL C01117 V=800.0 PL=0
MOVL C01118 V=800.0 PL=0
MOVL C01119 V=800.0 PL=0
MOVL C01120 V=800.0 PL=0
MOVL C01121 V=800.0 PL=0
MOVL C01122 V=800.0 PL=0
MOVL C01123 V=800.0 PL=0
MOVL C01124 V=800.0 PL=0
MOVL C01125 V=800.0 PL=0
MOVL C01126 V=800.0 PL=0
MOVL C01127 V=800.0 PL=0
MOVL C01128 V=800.0 PL=0
MOVL C01129 V=800.0 PL=0
MOVL C01130 V=800.0 PL=0
MOVL C01131 V=800.0 PL=0
MOVL C01132 V=800.0 PL=0
MOVL C01133 V=800.0 PL=0
MOVL C01134 V=800.0 PL=0
MOVL C01135 V=800.0 PL=0
MOVL C01136 V=800.0 PL=0
MOVL C01137 V=800.0 PL=0
MOVL C01138 V=800.0 PL=0
MOVL C01139 V=800.0 PL=0
MOVL C01140 V=800.0 PL=0
MOVL C01141 V=800.0 PL=0
MOVL C01142 V=800.0 PL=0
MOVL C01143 V=800.0 PL=0
MOVL C01144 V=800.0 PL=0
MOVL C01145 V=800.0 PL=0
MOVL C01146 V=800.0 PL=0
MOVL C01147 V=800.0 PL=0
MOVL C01148 V=800.0 PL=0
MOVL C01149 V=800.0 PL=0
MOVL C01150 V=800.0 PL=0
MOVL C01151 V=800.0 PL=0
MOVL C01152 V=800.0 PL=0
MOVL C01153 V=800.0 PL=0
MOVL C01154 V=800.0 PL=0
MOVL C01155 V=800.0 PL=0
MOVL C01156 V=800.0 PL=0
MOVL C01157 V=800.0 PL=0
MOVL C01158 V=800.0 PL=0
MOVL C01159 V=800.0 PL=0
MOVL C01160 V=800.0 PL=0
MOVL C01161 V=800.0 PL=0
MOVL C01162 V=800.0 PL=0
MOVL C01163 V=800.0 PL=0
MOVL C01164 V=800.0 PL=0
MOVL C01165 V=800.0 PL=0
MOVL C01166 V=800.0 PL=0
MOVL C01167 V=800.0 PL=0
MOVL C01168 V=800.0 PL=0
MOVL C01169 V=800.0 PL=0
MOVL C01170 V=800.0 PL=0
MOVL C01171 V=800.0 PL=0
MOVL C01172 V=800.0 PL=0
MOVL C01173 V=800.0 PL=0
MOVL C01174 V=800.0 PL=0
MOVL C01175 V=800.0 PL=0
MOVL C01176 V=800.0 PL=0
MOVL C01177 V=800.0 PL=0
MOVL C01178 V=800.0 PL=0
MOVL C01179 V=800.0 PL=0
MOVL C01180 V=800.0 PL=0
MOVL C01181 V=800.0 PL=0
MOVL C01182 V=800.0 PL=0
MOVL C01183 V=800.0 PL=0
MOVL C01184 V=800.0 PL=0
MOVL C01185 V=800.0 PL=0
MOVL C01186 V=800.0 PL=0
MOVL C01187 V=800.0 PL=0
MOVL C01188 V=800.0 PL=0
MOVL C01189 V=800.0 PL=0
MOVL C01190 V=800.0 PL=0
MOVL C01191 V=800.0 PL=0
MOVL C01192 V=800.0 PL=0
MOVL C01193 V=800.0 PL=0
MOVL C01194 V=800.0 PL=0
MOVL C01195 V=800.0 PL=0
MOVL C01196 V=800.0 PL=0
MOVL C01197 V=800.0 PL=0
MOVL C01198 V=800.0 PL=0
MOVL C01199 V=800.0 PL=0
MOVL C01200 V=800.0 PL=0
MOVL C01201 V=800.0 PL=0
MOVL C01202 V=800.0 PL=0
MOVL C01203 V=800.0 PL=0
MOVL C01204 V=800.0 PL=0
MOVL C01205 V=800.0 PL=0
MOVL C01206 V=800.0 PL=0
MOVL C01207 V=800.0 PL=0
MOVL C01208 V=800.0 PL=0
MOVL C01209 V=800.0 PL=0
MOVL C01210 V=800.0 PL=0
MOVL C01211 V=800.0 PL=0
MOVL C01212 V=800.0 PL=0
MOVL C01213 V=800.0 PL=0
MOVL C01214 V=800.0 PL=0
MOVL C01215 V=800.0 PL=0
MOVL C01216 V=800.0 PL=0
MOVL C01217 V=800.0 PL=0
MOVL C01218 V=800.0 PL=0
MOVL C01219 V=800.0 PL=0
MOVL C01220 V=800.0 PL=0
MOVL C01221 V=800.0 PL=0
MOVL C01222 V=800.0 PL=0
MOVL C01223 V=800.0 PL=0
MOVL C01224 V=800.0 PL=0
MOVL C01225 V=800.0 PL=0
MOVL C01226 V=800.0 PL=0
MOVL C01227 V=800.0 PL=0
MOVL C01228 V=800.0 PL=0
MOVL C01229 V=800.0 PL=0
MOVL C01230 V=800.0 PL=0
MOVL C01231 V=800.0 PL=0
MOVL C01232 V=800.0 PL=0
MOVL C01233 V=800.0 PL=0
MOVL C01234 V=800.0 PL=0
MOVL C01235 V=800.0 PL=0
MOVL C01236 V=800.0 PL=0
MOVL C01237 V=800.0 PL=0
MOVL C01238 V=800.0 PL=0
MOVL C01239 V=800.0 PL=0
MOVL C01240 V=800.0 PL=0
MOVL C01241 V=800.0 PL=0
MOVL C01242 V=800.0 PL=0
MOVL C01243 V=800.0 PL=0
MOVL C01244 V=800.0 PL=0
MOVL C01245 V=800.0 PL=0
MOVL C01246 V=800.0 PL=0
MOVL C01247 V=800.0 PL=0
MOVL C01248 V=800.0 PL=0
MOVL C01249 V=800.0 PL=0
MOVL C01250 V=800.0 PL=0
MOVL C01251 V=800.0 PL=0
MOVL C01252 V=800.0 PL=0
MOVL C01253 V=800.0 PL=0
MOVL C01254 V=800.0 PL=0
MOVL C01255 V=800.0 PL=0
MOVL C01256 V=800.0 PL=0
MOVL C01257 V=800.0 PL=0
MOVL C01258 V=800.0 PL=0
MOVL C01259 V=800.0 PL=0
MOVL C01260 V=800.0 PL=0
MOVL C01261 V=800.0 PL=0
MOVL C01262 V=800.0 PL=0
MOVL C01263 V=800.0 PL=0
MOVL C01264 V=800.0 PL=0
MOVL C01265 V=800.0 PL=0
MOVL C01266 V=800.0 PL=0
MOVL C01267 V=800.0 PL=0
MOVL C01268 V=800.0 PL=0
MOVL C01269 V=800.0 PL=0
MOVL C01270 V=800.0 PL=0
MOVL C01271 V=800.0 PL=0
MOVL C01272 V=800.0 PL=0
MOVL C01273 V=800.0 PL=0
MOVL C01274 V=800.0 PL=0
MOVL C01275 V=800.0 PL=0
MOVL C01276 V=800.0 PL=0
MOVL C01277 V=800.0 PL=0
MOVL C01278 V=800.0 PL=0
MOVL C01279 V=800.0 PL=0
MOVL C01280 V=800.0 PL=0
MOVL C01281 V=800.0 PL=0
MOVL C01282 V=800.0 PL=0
MOVL C01283 V=800.0 PL=0
MOVL C01284 V=800.0 PL=0
MOVL C01285 V=800.0 PL=0
MOVL C01286 V=800.0 PL=0
MOVL C01287 V=800.0 PL=0
MOVL C01288 V=800.0 PL=0
MOVL C01289 V=800.0 PL=0
MOVL C01290 V=800.0 PL=0
MOVL C01291 V=800.0 PL=0
MOVL C01292 V=800.0 PL=0
MOVL C01293 V=800.0 PL=0
MOVL C01294 V=800.0 PL=0
MOVL C01295 V=800.0 PL=0
MOVL C01296 V=800.0 PL=0
MOVL C01297 V=800.0 PL=0
MOVL C01298 V=800.0 PL=0
MOVL C01299 V=800.0 PL=0
MOVL C01300 V=800.0 PL=0
MOVL C01301 V=800.0 PL=0
MOVL C01302 V=800.0 PL=0
MOVL C01303 V=800.0 PL=0
MOVL C01304 V=800.0 PL=0
MOVL C01305 V=800.0 PL=0
MOVL C01306 V=800.0 PL=0
MOVL C01307 V=800.0 PL=0
MOVL C01308 V=800.0 PL=0
MOVL C01309 V=800.0 PL=0
MOVL C01310 V=800.0 PL=0
MOVL C01311 V=800.0 PL=0
MOVL C01312 V=800.0 PL=0
MOVL C01313 V=800.0 PL=0
MOVL C01314 V=800.0 PL=0
MOVL C01315 V=800.0 PL=0
MOVL C01316 V=800.0 PL=0
MOVL C01317 V=800.0 PL=0
MOVL C01318 V=800.0 PL=0
MOVL C01319 V=800.0 PL=0
MOVL C01320 V=800.0 PL=0
MOVL C01321 V=800.0 PL=0
MOVL C01322 V=800.0 PL=0
MOVL C01323 V=800.0 PL=0
MOVL C01324 V=800.0 PL=0
MOVL C01325 V=800.0 PL=0
MOVL C01326 V=800.0 PL=0
MOVL C01327 V=800.0 PL=0
MOVL C01328 V=800.0 PL=0
MOVL C01329 V=800.0 PL=0
MOVL C01330 V=800.0 PL=0
MOVL C01331 V=800.0 PL=0
MOVL C01332 V=800.0 PL=0
MOVL C01333 V=800.0 PL=0
MOVL C01334 V=800.0 PL=0
MOVL C01335 V=800.0 PL=0
MOVL C01336 V=800.0 PL=0
MOVL C01337 V=800.0 PL=0
MOVL C01338 V=800.0 PL=0
MOVL C01339 V=800.0 PL=0
MOVL C01340 V=800.0 PL=0
MOVL C01341 V=800.0 PL=0
MOVL C01342 V=800.0 PL=0
MOVL C01343 V=800.0 PL=0
MOVL C01344 V=800.0 PL=0
MOVL C01345 V=800.0 PL=0
MOVL C01346 V=800.0 PL=0
MOVL C01347 V=800.0 PL=0
MOVL C01348 V=800.0 PL=0
MOVL C01349 V=800.0 PL=0
MOVL C01350 V=800.0 PL=0
MOVL C01351 V=800.0 PL=0
MOVL C01352 V=800.0 PL=0
MOVL C01353 V=800.0 PL=0
MOVL C01354 V=800.0 PL=0
MOVL C01355 V=800.0 PL=0
MOVL C01356 V=800.0 PL=0
MOVL C01357 V=800.0 PL=0
MOVL C01358 V=800.0 PL=0
MOVL C01359 V=800.0 PL=0
MOVL C01360 V=800.0 PL=0
MOVL C01361 V=800.0 PL=0
MOVL C01362 V=800.0 PL=0
MOVL C01363 V=800.0 PL=0
MOVL C01364 V=800.0 PL=0
MOVL C01365 V=800.0 PL=0
MOVL C01366 V=800.0 PL=0
MOVL C01367 V=800.0 PL=0
MOVL C01368 V=800.0 PL=0
MOVL C01369 V=800.0 PL=0
MOVL C01370 V=800.0 PL=0
MOVL C01371 V=800.0 PL=0
MOVL C01372 V=800.0 PL=0
MOVL C01373 V=800.0 PL=0
MOVL C01374 V=800.0 PL=0
MOVL C01375 V=800.0 PL=0
MOVL C01376 V=800.0 PL=0
MOVL C01377 V=800.0 PL=0
MOVL C01378 V=800.0 PL=0
MOVL C01379 V=800.0 PL=0
MOVL C01380 V=800.0 PL=0
MOVL C01381 V=800.0 PL=0
MOVL C01382 V=800.0 PL=0
MOVL C01383 V=800.0 PL=0
MOVL C01384 V=800.0 PL=0
MOVL C01385 V=800.0 PL=0
MOVL C01386 V=800.0 PL=0
MOVL C01387 V=800.0 PL=0
MOVL C01388 V=800.0 PL=0
MOVL C01389 V=800.0 PL=0
MOVL C01390 V=800.0 PL=0
MOVL C01391 V=800.0 PL=0
MOVL C01392 V=800.0 PL=0
MOVL C01393 V=800.0 PL=0
MOVL C01394 V=800.0 PL=0
MOVL C01395 V=800.0 PL=0
MOVL C01396 V=800.0 PL=0
MOVL C01397 V=800.0 PL=0
MOVL C01398 V=800.0 PL=0
MOVL C01399 V=800.0 PL=0
MOVL C01400 V=800.0 PL=0
MOVL C01401 V=800.0 PL=0
MOVL C01402 V=800.0 PL=0
MOVL C01403 V=800.0 PL=0
MOVL C01404 V=800.0 PL=0
MOVL C01405 V=800.0 PL=0
MOVL C01406 V=800.0 PL=0
MOVL C01407 V=800.0 PL=0
MOVL C01408 V=800.0 PL=0
MOVL C01409 V=800.0 PL=0
MOVL C01410 V=800.0 PL=0
MOVL C01411 V=800.0 PL=0
MOVL C01412 V=800.0 PL=0
MOVL C01413 V=800.0 PL=0
MOVL C01414 V=800.0 PL=0
MOVL C01415 V=800.0 PL=0
MOVL C01416 V=800.0 PL=0
MOVL C01417 V=800.0 PL=0
MOVL C01418 V=800.0 PL=0
MOVL C01419 V=800.0 PL=0
MOVL C01420 V=800.0 PL=0
MOVL C01421 V=800.0 PL=0
MOVL C01422 V=800.0 PL=0
MOVL C01423 V=800.0 PL=0
MOVL C01424 V=800.0 PL=0
MOVL C01425 V=800.0 PL=0
MOVL C01426 V=800.0 PL=0
MOVL C01427 V=800.0 PL=0
MOVL C01428 V=800.0 PL=0
MOVL C01429 V=800.0 PL=0
MOVL C01430 V=800.0 PL=0
MOVL C01431 V=800.0 PL=0
MOVL C01432 V=800.0 PL=0
MOVL C01433 V=800.0 PL=0
MOVL C01434 V=800.0 PL=0
MOVL C01435 V=800.0 PL=0
MOVL C01436 V=800.0 PL=0
MOVL C01437 V=800.0 PL=0
MOVL C01438 V=800.0 PL=0
MOVL C01439 V=800.0 PL=0
MOVL C01440 V=800.0 PL=0
MOVL C01441 V=800.0 PL=0
MOVL C01442 V=800.0 PL=0
MOVL C01443 V=800.0 PL=0
MOVL C01444 V=800.0 PL=0
MOVL C01445 V=800.0 PL=0
MOVL C01446 V=800.0 PL=0
MOVL C01447 V=800.0 PL=0
MOVL C01448 V=800.0 PL=0
MOVL C01449 V=800.0 PL=0
MOVL C01450 V=800.0 PL=0
MOVL C01451 V=800.0 PL=0
MOVL C01452 V=800.0 PL=0
MOVL C01453 V=800.0 PL=0
MOVL C01454 V=800.0 PL=0
MOVL C01455 V=800.0 PL=0
MOVL C01456 V=800.0 PL=0
MOVL C01457 V=800.0 PL=0
MOVL C01458 V=800.0 PL=0
MOVL C01459 V=800.0 PL=0
MOVL C01460 V=800.0 PL=0
MOVL C01461 V=800.0 PL=0
MOVL C01462 V=800.0 PL=0
MOVL C01463 V=800.0 PL=0
MOVL C01464 V=800.0 PL=0
MOVL C01465 V=800.0 PL=0
MOVL C01466 V=800.0 PL=0
MOVL C01467 V=800.0 PL=0
MOVL C01468 V=800.0 PL=0
MOVL C01469 V=800.0 PL=0
MOVL C01470 V=800.0 PL=0
MOVL C01471 V=800.0 PL=0
MOVL C01472 V=800.0 PL=0
MOVL C01473 V=800.0 PL=0
MOVL C01474 V=800.0 PL=0
MOVL C01475 V=800.0 PL=0
MOVL C01476 V=800.0 PL=0
MOVL C01477 V=800.0 PL=0
MOVL C01478 V=800.0 PL=0
MOVL C01479 V=800.0 PL=0
MOVL C01480 V=800.0 PL=0
MOVL C01481 V=800.0 PL=0
MOVL C01482 V=800.0 PL=0
MOVL C01483 V=800.0 PL=0
MOVL C01484 V=800.0 PL=0
MOVL C01485 V=800.0 PL=0
MOVL C01486 V=800.0 PL=0
MOVL C01487 V=800.0 PL=0
MOVL C01488 V=800.0 PL=0
MOVL C01489 V=800.0 PL=0
MOVL C01490 V=800.0 PL=0
MOVL C01491 V=800.0 PL=0
MOVL C01492 V=800.0 PL=0
MOVL C01493 V=800.0 PL=0
MOVL C01494 V=800.0 PL=0
MOVL C01495 V=800.0 PL=0
MOVL C01496 V=800.0 PL=0
MOVL C01497 V=800.0 PL=0
MOVL C01498 V=800.0 PL=0
MOVL C01499 V=800.0 PL=0
MOVL C01500 V=800.0 PL=0
MOVL C01501 V=800.0 PL=0
MOVL C01502 V=800.0 PL=0
MOVL C01503 V=800.0 PL=0
MOVL C01504 V=800.0 PL=0
MOVL C01505 V=800.0 PL=0
MOVL C01506 V=800.0 PL=0
MOVL C01507 V=800.0 PL=0
MOVL C01508 V=800.0 PL=0
MOVL C01509 V=800.0 PL=0
MOVL C01510 V=800.0 PL=0
MOVL C01511 V=800.0 PL=0
MOVL C01512 V=800.0 PL=0
MOVL C01513 V=800.0 PL=0
MOVL C01514 V=800.0 PL=0
MOVL C01515 V=800.0 PL=0
MOVL C01516 V=800.0 PL=0
MOVL C01517 V=800.0 PL=0
MOVL C01518 V=800.0 PL=0
MOVL C01519 V=800.0 PL=0
MOVL C01520 V=800.0 PL=0
MOVL C01521 V=800.0 PL=0
MOVL C01522 V=800.0 PL=0
MOVL C01523 V=800.0 PL=0
MOVL C01524 V=800.0 PL=0
MOVL C01525 V=800.0 PL=0
MOVL C01526 V=800.0 PL=0
MOVL C01527 V=800.0 PL=0
MOVL C01528 V=800.0 PL=0
MOVL C01529 V=800.0 PL=0
MOVL C01530 V=800.0 PL=0
MOVL C01531 V=800.0 PL=0
MOVL C01532 V=800.0 PL=0
MOVL C01533 V=800.0 PL=0
MOVL C01534 V=800.0 PL=0
MOVL C01535 V=800.0 PL=0
MOVL C01536 V=800.0 PL=0
MOVL C01537 V=800.0 PL=0
MOVL C01538 V=800.0 PL=0
MOVL C01539 V=800.0 PL=0
MOVL C01540 V=800.0 PL=0
MOVL C01541 V=800.0 PL=0
MOVL C01542 V=800.0 PL=0
MOVL C01543 V=800.0 PL=0
MOVL C01544 V=800.0 PL=0
MOVL C01545 V=800.0 PL=0
MOVL C01546 V=800.0 PL=0
MOVL C01547 V=800.0 PL=0
MOVL C01548 V=800.0 PL=0
MOVL C01549 V=800.0 PL=0
MOVL C01550 V=800.0 PL=0
MOVL C01551 V=800.0 PL=0
MOVL C01552 V=800.0 PL=0
MOVL C01553 V=800.0 PL=0
MOVL C01554 V=800.0 PL=0
MOVL C01555 V=800.0 PL=0
MOVL C01556 V=800.0 PL=0
MOVL C01557 V=800.0 PL=0
MOVL C01558 V=800.0 PL=0
MOVL C01559 V=800.0 PL=0
MOVL C01560 V=800.0 PL=0
MOVL C01561 V=800.0 PL=0
MOVL C01562 V=800.0 PL=0
MOVL C01563 V=800.0 PL=0
MOVL C01564 V=800.0 PL=0
MOVL C01565 V=800.0 PL=0
MOVL C01566 V=800.0 PL=0
MOVL C01567 V=800.0 PL=0
MOVL C01568 V=800.0 PL=0
MOVL C01569 V=800.0 PL=0
MOVL C01570 V=800.0 PL=0
MOVL C01571 V=800.0 PL=0
MOVL C01572 V=800.0 PL=0
MOVL C01573 V=800.0 PL=0
MOVL C01574 V=800.0 PL=0
MOVL C01575 V=800.0 PL=0
MOVL C01576 V=800.0 PL=0
MOVL C01577 V=800.0 PL=0
MOVL C01578 V=800.0 PL=0
MOVL C01579 V=800.0 PL=0
MOVL C01580 V=800.0 PL=0
MOVL C01581 V=800.0 PL=0
MOVL C01582 V=800.0 PL=0
MOVL C01583 V=800.0 PL=0
MOVL C01584 V=800.0 PL=0
MOVL C01585 V=800.0 PL=0
MOVL C01586 V=800.0 PL=0
MOVL C01587 V=800.0 PL=0
MOVL C01588 V=800.0 PL=0
MOVL C01589 V=800.0 PL=0
MOVL C01590 V=800.0 PL=0
MOVL C01591 V=800.0 PL=0
MOVL C01592 V=800.0 PL=0
MOVL C01593 V=800.0 PL=0
MOVL C01594 V=800.0 PL=0
MOVL C01595 V=800.0 PL=0
MOVL C01596 V=800.0 PL=0
MOVL C01597 V=800.0 PL=0
MOVL C01598 V=800.0 PL=0
MOVL C01599 V=800.0 PL=0
MOVL C01600 V=800.0 PL=0
MOVL C01601 V=800.0 PL=0
MOVL C01602 V=800.0 PL=0
MOVL C01603 V=800.0 PL=0
MOVL C01604 V=800.0 PL=0
MOVL C01605 V=800.0 PL=0
MOVL C01606 V=800.0 PL=0
MOVL C01607 V=800.0 PL=0
MOVL C01608 V=800.0 PL=0
MOVL C01609 V=800.0 PL=0
MOVL C01610 V=800.0 PL=0
MOVL C01611 V=800.0 PL=0
MOVL C01612 V=800.0 PL=0
MOVL C01613 V=800.0 PL=0
MOVL C01614 V=800.0 PL=0
MOVL C01615 V=800.0 PL=0
MOVL C01616 V=800.0 PL=0
MOVL C01617 V=800.0 PL=0
MOVL C01618 V=800.0 PL=0
MOVL C01619 V=800.0 PL=0
MOVL C01620 V=800.0 PL=0
MOVL C01621 V=800.0 PL=0
MOVL C01622 V=800.0 PL=0
MOVL C01623 V=800.0 PL=0
MOVL C01624 V=800.0 PL=0
MOVL C01625 V=800.0 PL=0
MOVL C01626 V=800.0 PL=0
MOVL C01627 V=800.0 PL=0
MOVL C01628 V=800.0 PL=0
MOVL C01629 V=800.0 PL=0
MOVL C01630 V=800.0 PL=0
MOVL C01631 V=800.0 PL=0
MOVL C01632 V=800.0 PL=0
MOVL C01633 V=800.0 PL=0
MOVL C01634 V=800.0 PL=0
MOVL C01635 V=800.0 PL=0
MOVL C01636 V=800.0 PL=0
MOVL C01637 V=800.0 PL=0
MOVL C01638 V=800.0 PL=0
MOVL C01639 V=800.0 PL=0
MOVL C01640 V=800.0 PL=0
MOVL C01641 V=800.0 PL=0
MOVL C01642 V=800.0 PL=0
MOVL C01643 V=800.0 PL=0
MOVL C01644 V=800.0 PL=0
MOVL C01645 V=800.0 PL=0
MOVL C01646 V=800.0 PL=0
MOVL C01647 V=800.0 PL=0
MOVL C01648 V=800.0 PL=0
MOVL C01649 V=800.0 PL=0
MOVL C01650 V=800.0 PL=0
MOVL C01651 V=800.0 PL=0
MOVL C01652 V=800.0 PL=0
MOVL C01653 V=800.0 PL=0
MOVL C01654 V=800.0 PL=0
MOVL C01655 V=800.0 PL=0
MOVL C01656 V=800.0 PL=0
MOVL C01657 V=800.0 PL=0
MOVL C01658 V=800.0 PL=0
MOVL C01659 V=800.0 PL=0
MOVL C01660 V=800.0 PL=0
MOVL C01661 V=800.0 PL=0
MOVL C01662 V=800.0 PL=0
MOVL C01663 V=800.0 PL=0
MOVL C01664 V=800.0 PL=0
MOVL C01665 V=800.0 PL=0
MOVL C01666 V=800.0 PL=0
MOVL C01667 V=800.0 PL=0
MOVL C01668 V=800.0 PL=0
MOVL C01669 V=800.0 PL=0
MOVL C01670 V=800.0 PL=0
MOVL C01671 V=800.0 PL=0
MOVL C01672 V=800.0 PL=0
MOVL C01673 V=800.0 PL=0
MOVL C01674 V=800.0 PL=0
MOVL C01675 V=800.0 PL=0
MOVL C01676 V=800.0 PL=0
MOVL C01677 V=800.0 PL=0
MOVL C01678 V=800.0 PL=0
MOVL C01679 V=800.0 PL=0
MOVL C01680 V=800.0 PL=0
MOVL C01681 V=800.0 PL=0
MOVL C01682 V=800.0 PL=0
MOVL C01683 V=800.0 PL=0
MOVL C01684 V=800.0 PL=0
MOVL C01685 V=800.0 PL=0
MOVL C01686 V=800.0 PL=0
MOVL C01687 V=800.0 PL=0
MOVL C01688 V=800.0 PL=0
MOVL C01689 V=800.0 PL=0
MOVL C01690 V=800.0 PL=0
MOVL C01691 V=800.0 PL=0
MOVL C01692 V=800.0 PL=0
MOVL C01693 V=800.0 PL=0
MOVL C01694 V=800.0 PL=0
MOVL C01695 V=800.0 PL=0
MOVL C01696 V=800.0 PL=0
MOVL C01697 V=800.0 PL=0
MOVL C01698 V=800.0 PL=0
MOVL C01699 V=800.0 PL=0
MOVL C01700 V=800.0 PL=0
MOVL C01701 V=800.0 PL=0
MOVL C01702 V=800.0 PL=0
MOVL C01703 V=800.0 PL=0
MOVL C01704 V=800.0 PL=0
MOVL C01705 V=800.0 PL=0
MOVL C01706 V=800.0 PL=0
MOVL C01707 V=800.0 PL=0
MOVL C01708 V=800.0 PL=0
MOVL C01709 V=800.0 PL=0
MOVL C01710 V=800.0 PL=0
MOVL C01711 V=800.0 PL=0
MOVL C01712 V=800.0 PL=0
MOVL C01713 V=800.0 PL=0
MOVL C01714 V=800.0 PL=0
MOVL C01715 V=800.0 PL=0
MOVL C01716 V=800.0 PL=0
MOVL C01717 V=800.0 PL=0
MOVL C01718 V=800.0 PL=0
MOVL C01719 V=800.0 PL=0
MOVL C01720 V=800.0 PL=0
MOVL C01721 V=800.0 PL=0
MOVL C01722 V=800.0 PL=0
MOVL C01723 V=800.0 PL=0
MOVL C01724 V=800.0 PL=0
MOVL C01725 V=800.0 PL=0
MOVL C01726 V=800.0 PL=0
MOVL C01727 V=800.0 PL=0
MOVL C01728 V=800.0 PL=0
MOVL C01729 V=800.0 PL=0
MOVL C01730 V=800.0 PL=0
MOVL C01731 V=800.0 PL=0
MOVL C01732 V=800.0 PL=0
MOVL C01733 V=800.0 PL=0
MOVL C01734 V=800.0 PL=0
MOVL C01735 V=800.0 PL=0
MOVL C01736 V=800.0 PL=0
MOVL C01737 V=800.0 PL=0
MOVL C01738 V=800.0 PL=0
MOVL C01739 V=800.0 PL=0
MOVL C01740 V=800.0 PL=0
MOVL C01741 V=800.0 PL=0
MOVL C01742 V=800.0 PL=0
MOVL C01743 V=800.0 PL=0
MOVL C01744 V=800.0 PL=0
MOVL C01745 V=800.0 PL=0
MOVL C01746 V=800.0 PL=0
MOVL C01747 V=800.0 PL=0
MOVL C01748 V=800.0 PL=0
MOVL C01749 V=800.0 PL=0
MOVL C01750 V=800.0 PL=0
MOVL C01751 V=800.0 PL=0
MOVL C01752 V=800.0 PL=0
MOVL C01753 V=800.0 PL=0
MOVL C01754 V=800.0 PL=0
MOVL C01755 V=800.0 PL=0
MOVL C01756 V=800.0 PL=0
MOVL C01757 V=800.0 PL=0
MOVL C01758 V=800.0 PL=0
MOVL C01759 V=800.0 PL=0
MOVL C01760 V=800.0 PL=0
MOVL C01761 V=800.0 PL=0
MOVL C01762 V=800.0 PL=0
MOVL C01763 V=800.0 PL=0
MOVL C01764 V=800.0 PL=0
MOVL C01765 V=800.0 PL=0
MOVL C01766 V=800.0 PL=0
MOVL C01767 V=800.0 PL=0
MOVL C01768 V=800.0 PL=0
MOVL C01769 V=800.0 PL=0
MOVL C01770 V=800.0 PL=0
MOVL C01771 V=800.0 PL=0
MOVL C01772 V=800.0 PL=0
MOVL C01773 V=800.0 PL=0
MOVL C01774 V=800.0 PL=0
MOVL C01775 V=800.0 PL=0
MOVL C01776 V=800.0 PL=0
MOVL C01777 V=800.0 PL=0
MOVL C01778 V=800.0 PL=0
MOVL C01779 V=800.0 PL=0
MOVL C01780 V=800.0 PL=0
MOVL C01781 V=800.0 PL=0
MOVL C01782 V=800.0 PL=0
MOVL C01783 V=800.0 PL=0
MOVL C01784 V=800.0 PL=0
MOVL C01785 V=800.0 PL=0
MOVL C01786 V=800.0 PL=0
MOVL C01787 V=800.0 PL=0
MOVL C01788 V=800.0 PL=0
MOVL C01789 V=800.0 PL=0
MOVL C01790 V=800.0 PL=0
MOVL C01791 V=800.0 PL=0
MOVL C01792 V=800.0 PL=0
MOVL C01793 V=800.0 PL=0
MOVL C01794 V=800.0 PL=0
MOVL C01795 V=800.0 PL=0
MOVL C01796 V=800.0 PL=0
MOVL C01797 V=800.0 PL=0
MOVL C01798 V=800.0 PL=0
MOVL C01799 V=800.0 PL=0
MOVL C01800 V=800.0 PL=0
MOVL C01801 V=800.0 PL=0
MOVL C01802 V=800.0 PL=0
MOVL C01803 V=800.0 PL=0
MOVL C01804 V=800.0 PL=0
MOVL C01805 V=800.0 PL=0
MOVL C01806 V=800.0 PL=0
MOVL C01807 V=800.0 PL=0
MOVL C01808 V=800.0 PL=0
MOVL C01809 V=800.0 PL=0
MOVL C01810 V=800.0 PL=0
MOVL C01811 V=800.0 PL=0
MOVL C01812 V=800.0 PL=0
MOVL C01813 V=800.0 PL=0
MOVL C01814 V=800.0 PL=0
MOVL C01815 V=800.0 PL=0
MOVL C01816 V=800.0 PL=0
MOVL C01817 V=800.0 PL=0
MOVL C01818 V=800.0 PL=0
MOVL C01819 V=800.0 PL=0
MOVL C01820 V=800.0 PL=0
MOVL C01821 V=800.0 PL=0
MOVL C01822 V=800.0 PL=0
MOVL C01823 V=800.0 PL=0
MOVL C01824 V=800.0 PL=0
MOVL C01825 V=800.0 PL=0
MOVL C01826 V=800.0 PL=0
MOVL C01827 V=800.0 PL=0
MOVL C01828 V=800.0 PL=0
MOVL C01829 V=800.0 PL=0
MOVL C01830 V=800.0 PL=0
MOVL C01831 V=800.0 PL=0
MOVL C01832 V=800.0 PL=0
MOVL C01833 V=800.0 PL=0
MOVL C01834 V=800.0 PL=0
MOVL C01835 V=800.0 PL=0
MOVL C01836 V=800.0 PL=0
MOVL C01837 V=800.0 PL=0
MOVL C01838 V=800.0 PL=0
MOVL C01839 V=800.0 PL=0
MOVL C01840 V=800.0 PL=0
MOVL C01841 V=800.0 PL=0
MOVL C01842 V=800.0 PL=0
MOVL C01843 V=800.0 PL=0
MOVL C01844 V=800.0 PL=0
MOVL C01845 V=800.0 PL=0
MOVL C01846 V=800.0 PL=0
MOVL C01847 V=800.0 PL=0
MOVL C01848 V=800.0 PL=0
MOVL C01849 V=800.0 PL=0
MOVL C01850 V=800.0 PL=0
MOVL C01851 V=800.0 PL=0
MOVL C01852 V=800.0 PL=0
MOVL C01853 V=800.0 PL=0
MOVL C01854 V=800.0 PL=0
MOVL C01855 V=800.0 PL=0
MOVL C01856 V=800.0 PL=0
MOVL C01857 V=800.0 PL=0
MOVL C01858 V=800.0 PL=0
MOVL C01859 V=800.0 PL=0
MOVL C01860 V=800.0 PL=0
MOVL C01861 V=800.0 PL=0
MOVL C01862 V=800.0 PL=0
MOVL C01863 V=800.0 PL=0
MOVL C01864 V=800.0 PL=0
MOVL C01865 V=800.0 PL=0
MOVL C01866 V=800.0 PL=0
MOVL C01867 V=800.0 PL=0
MOVL C01868 V=800.0 PL=0
MOVL C01869 V=800.0 PL=0
MOVL C01870 V=800.0 PL=0
MOVL C01871 V=800.0 PL=0
MOVL C01872 V=800.0 PL=0
MOVL C01873 V=800.0 PL=0
MOVL C01874 V=800.0 PL=0
MOVL C01875 V=800.0 PL=0
MOVL C01876 V=800.0 PL=0
MOVL C01877 V=800.0 PL=0
MOVL C01878 V=800.0 PL=0
MOVL C01879 V=800.0 PL=0
MOVL C01880 V=800.0 PL=0
MOVL C01881 V=800.0 PL=0
MOVL C01882 V=800.0 PL=0
MOVL C01883 V=800.0 PL=0
MOVL C01884 V=800.0 PL=0
MOVL C01885 V=800.0 PL=0
MOVL C01886 V=800.0 PL=0
MOVL C01887 V=800.0 PL=0
MOVL C01888 V=800.0 PL=0
MOVL C01889 V=800.0 PL=0
MOVL C01890 V=800.0 PL=0
MOVL C01891 V=800.0 PL=0
MOVL C01892 V=800.0 PL=0
MOVL C01893 V=800.0 PL=0
MOVL C01894 V=800.0 PL=0
MOVL C01895 V=800.0 PL=0
MOVL C01896 V=800.0 PL=0
MOVL C01897 V=800.0 PL=0
MOVL C01898 V=800.0 PL=0
MOVL C01899 V=800.0 PL=0
MOVL C01900 V=800.0 PL=0
MOVL C01901 V=800.0 PL=0
MOVL C01902 V=800.0 PL=0
MOVL C01903 V=800.0 PL=0
MOVL C01904 V=800.0 PL=0
MOVL C01905 V=800.0 PL=0
MOVL C01906 V=800.0 PL=0
MOVL C01907 V=800.0 PL=0
MOVL C01908 V=800.0 PL=0
MOVL C01909 V=800.0 PL=0
MOVL C01910 V=800.0 PL=0
MOVL C01911 V=800.0 PL=0
MOVL C01912 V=800.0 PL=0
MOVL C01913 V=800.0 PL=0
MOVL C01914 V=800.0 PL=0
MOVL C01915 V=800.0 PL=0
MOVL C01916 V=800.0 PL=0
MOVL C01917 V=800.0 PL=0
MOVL C01918 V=800.0 PL=0
MOVL C01919 V=800.0 PL=0
MOVL C01920 V=800.0 PL=0
MOVL C01921 V=800.0 PL=0
MOVL C01922 V=800.0 PL=0
MOVL C01923 V=800.0 PL=0
MOVL C01924 V=800.0 PL=0
MOVL C01925 V=800.0 PL=0
MOVL C01926 V=800.0 PL=0
MOVL C01927 V=800.0 PL=0
MOVL C01928 V=800.0 PL=0
MOVL C01929 V=800.0 PL=0
MOVL C01930 V=800.0 PL=0
MOVL C01931 V=800.0 PL=0
MOVL C01932 V=800.0 PL=0
MOVL C01933 V=800.0 PL=0
MOVL C01934 V=800.0 PL=0
MOVL C01935 V=800.0 PL=0
MOVL C01936 V=800.0 PL=0
MOVL C01937 V=800.0 PL=0
MOVL C01938 V=800.0 PL=0
MOVL C01939 V=800.0 PL=0
MOVL C01940 V=800.0 PL=0
MOVL C01941 V=800.0 PL=0
MOVL C01942 V=800.0 PL=0
MOVL C01943 V=800.0 PL=0
MOVL C01944 V=800.0 PL=0
MOVL C01945 V=800.0 PL=0
MOVL C01946 V=800.0 PL=0
MOVL C01947 V=800.0 PL=0
MOVL C01948 V=800.0 PL=0
MOVL C01949 V=800.0 PL=0
MOVL C01950 V=800.0 PL=0
MOVL C01951 V=800.0 PL=0
MOVL C01952 V=800.0 PL=0
MOVL C01953 V=800.0 PL=0
MOVL C01954 V=800.0 PL=0
MOVL C01955 V=800.0 PL=0
MOVL C01956 V=800.0 PL=0
MOVL C01957 V=800.0 PL=0
MOVL C01958 V=800.0 PL=0
MOVL C01959 V=800.0 PL=0
MOVL C01960 V=800.0 PL=0
MOVL C01961 V=800.0 PL=0
MOVL C01962 V=800.0 PL=0
MOVL C01963 V=800.0 PL=0
MOVL C01964 V=800.0 PL=0
MOVL C01965 V=800.0 PL=0
MOVL C01966 V=800.0 PL=0
MOVL C01967 V=800.0 PL=0
MOVL C01968 V=800.0 PL=0
MOVL C01969 V=800.0 PL=0
MOVL C01970 V=800.0 PL=0
MOVL C01971 V=800.0 PL=0
MOVL C01972 V=800.0 PL=0
MOVL C01973 V=800.0 PL=0
MOVL C01974 V=800.0 PL=0
MOVL C01975 V=800.0 PL=0
MOVL C01976 V=800.0 PL=0
MOVL C01977 V=800.0 PL=0
MOVL C01978 V=800.0 PL=0
MOVL C01979 V=800.0 PL=0
MOVL C01980 V=800.0 PL=0
MOVL C01981 V=800.0 PL=0
MOVL C01982 V=800.0 PL=0
MOVL C01983 V=800.0 PL=0
MOVL C01984 V=800.0 PL=0
MOVL C01985 V=800.0 PL=0
MOVL C01986 V=800.0 PL=0
MOVL C01987 V=800.0 PL=0
MOVL C01988 V=800.0 PL=0
MOVL C01989 V=800.0 PL=0
MOVL C01990 V=800.0 PL=0
MOVL C01991 V=800.0 PL=0
MOVL C01992 V=800.0 PL=0
MOVL C01993 V=800.0 PL=0
MOVL C01994 V=800.0 PL=0
MOVL C01995 V=800.0 PL=0
MOVL C01996 V=800.0 PL=0
MOVL C01997 V=800.0 PL=0
MOVL C01998 V=800.0 PL=0
MOVL C01999 V=800.0 PL=0
MOVL C02000 V=800.0 PL=0
MOVL C02001 V=800.0 PL=0
MOVL C02002 V=800.0 PL=0
MOVL C02003 V=800.0 PL=0
MOVL C02004 V=800.0 PL=0
MOVL C02005 V=800.0 PL=0
MOVL C02006 V=800.0 PL=0
MOVL C02007 V=800.0 PL=0
MOVL C02008 V=800.0 PL=0
MOVL C02009 V=800.0 PL=0
MOVL C02010 V=800.0 PL=0
MOVL C02011 V=800.0 PL=0
MOVL C02012 V=800.0 PL=0
MOVL C02013 V=800.0 PL=0
MOVL C02014 V=800.0 PL=0
MOVL C02015 V=800.0 PL=0
MOVL C02016 V=800.0 PL=0
MOVL C02017 V=800.0 PL=0
MOVL C02018 V=800.0 PL=0
MOVL C02019 V=800.0 PL=0
MOVL C02020 V=800.0 PL=0
MOVL C02021 V=800.0 PL=0
MOVL C02022 V=800.0 PL=0
MOVL C02023 V=800.0 PL=0
MOVL C02024 V=800.0 PL=0
MOVL C02025 V=800.0 PL=0
MOVL C02026 V=800.0 PL=0
MOVL C02027 V=800.0 PL=0
MOVL C02028 V=800.0 PL=0
MOVL C02029 V=800.0 PL=0
MOVL C02030 V=800.0 PL=0
MOVL C02031 V=800.0 PL=0
MOVL C02032 V=800.0 PL=0
MOVL C02033 V=800.0 PL=0
MOVL C02034 V=800.0 PL=0
MOVL C02035 V=800.0 PL=0
MOVL C02036 V=800.0 PL=0
MOVL C02037 V=800.0 PL=0
MOVL C02038 V=800.0 PL=0
MOVL C02039 V=800.0 PL=0
MOVL C02040 V=800.0 PL=0
MOVL C02041 V=800.0 PL=0
MOVL C02042 V=800.0 PL=0
MOVL C02043 V=800.0 PL=0
MOVL C02044 V=800.0 PL=0
MOVL C02045 V=800.0 PL=0
MOVL C02046 V=800.0 PL=0
MOVL C02047 V=800.0 PL=0
